RoboDK station: main for aircraft.rdk

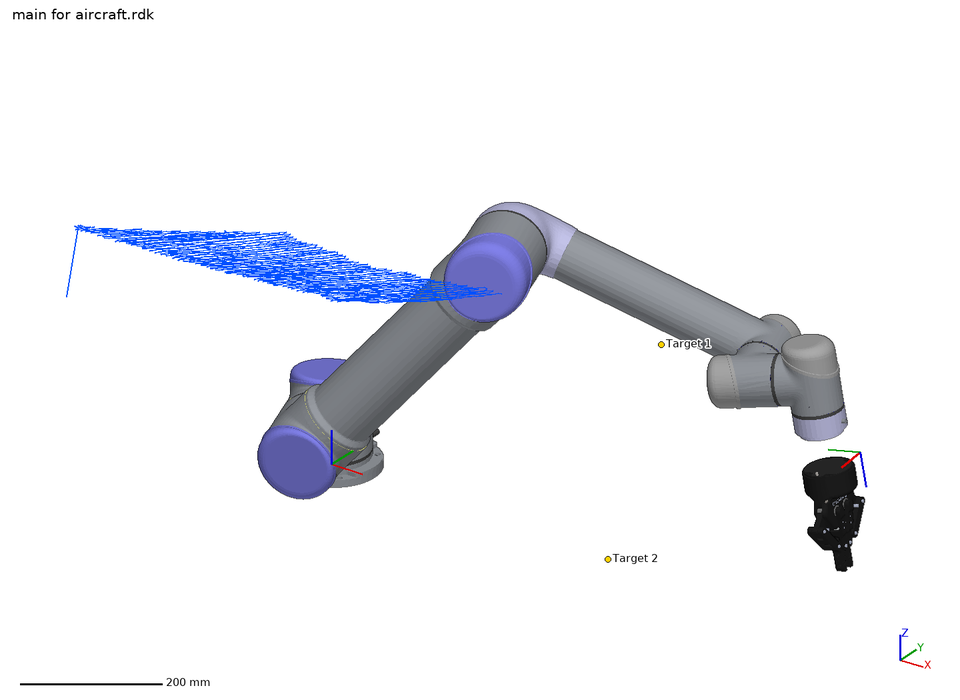
[picture v0: the station drawn from its stored meshes, robots at their saved joint values, targets as dots, program paths as lines]
Station main. Poses are relative to the parent item; angles as X-Y-Z fixed-axis rotations.
  - frame UR5 Base at (0, 0, 0) mm
    - robot UR5: 6 axes, payload 5 kg, reach 850 mm, repeatability 0.1 mm, weight 18.4 kg
        modified DH rows (alpha deg, a mm, theta deg, d mm): 0, 0, 0, 89.2; 90, 0, 180, 0; 0, 425, 0, 0; 0, 392.43, 0, 109; -90, 0, 0, 93.65; 90, 0, 180, 82
        joint limits [-360, -360, -360, -360, -360, -360] to [360, 360, 360, 360, 360, 360]; home [0, -90, -90, 0, 90, 0]; saved at [19.212, -130.821, -70.481, -59.3, 88.748, 13.688]
      - tool Gripper RobotiQ 85 Fully closed, TCP at (0, 0, 221.6) mm, size 121.5 x 75 x 160.2 mm
      - frame Object at (0, -58.4, 27.12) mm
        - object cloud_2 at (0, 0, 0) mm
    - target Target 1 (Cartesian target) at (643.45, -109, 411.64) mm, rotated rx -90 ry 0 rz -90 deg; joints [0, -90, -120, 30, 90, 0] of UR5
    - target Target 2 (Cartesian target) at (518.34, -61.08, 20.7) mm, rotated rx -149.99 ry -0.01 rz -84.67 deg; joints [5.34, -89.99, -135, -15, 89.99, 0] of UR5
  - machining project Path1 settings: rotZ(0) | rotX(0)*rotY(0) | rotZ(0)
  - program Path1 (2180 instructions, listed below)
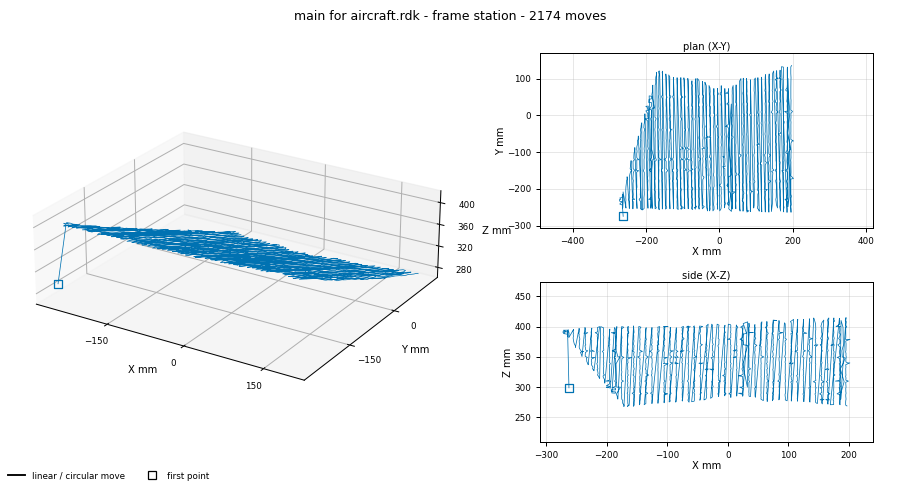
[picture p0: tool path of main for aircraft.rdk in frame station, 2174 of 2174 moves have a stored position in this frame; points joined in program order, loops and branches not executed]

--- program Path1 (robot UR5) ---
  Smooth(10)
  Set Ref.: UR5 Base
  Set Tool: Gripper RobotiQ 85 Fully closed
  Show Gripper RobotiQ 85 Fully closed
  Set speed (1000.0 mm/s)
  MoveJ 1 to (-262.02, -274.89, 298.94) mm, rotated rx -17.88 ry -1.25 rz 0.4 deg; joints [23.669, -136.733, -44.176, -77.159, 87.449, 17.927]
  MoveL 2 to (-262.02, -274.89, 298.94) mm, rotated rx -17.88 ry -1.25 rz 0.4 deg; joints [23.669, -136.733, -44.176, -77.159, 87.449, 17.927]
  MoveL 3 to (-264.31, -244.19, 394.09) mm, rotated rx -17.88 ry -1.25 rz 0.4 deg; joints [23.356, -142.512, -47.963, -67.579, 87.514, 17.62]
  MoveL 4 to (-264.31, -244.19, 394.09) mm, rotated rx -17.88 ry -1.25 rz 0.4 deg; joints [23.356, -142.512, -47.963, -67.579, 87.514, 17.62]
  Set speed (15.0 mm/s)
  MoveL 5 to (-271.37, -241.29, 394) mm, rotated rx -17.59 ry -0.18 rz 0.06 deg; joints [24.315, -142.277, -48.615, -67.291, 86.159, 18.561]
  MoveL 6 to (-265.21, -234.85, 391.18) mm, rotated rx -18.34 ry -0.72 rz 0.24 deg; joints [23.771, -141.372, -50.184, -67.121, 87.044, 18.065]
  MoveL 7 to (-271.75, -233.48, 391.83) mm, rotated rx -17.96 ry 0.25 rz -0.08 deg; joints [24.636, -141.351, -50.461, -66.885, 85.792, 18.911]
  MoveL 8 to (-271.9, -228.84, 390.33) mm, rotated rx -18.1 ry 0.31 rz -0.1 deg; joints [24.767, -140.701, -51.764, -66.391, 85.742, 19.05]
  MoveL 9 to (-268.61, -228.64, 390) mm, rotated rx -18.14 ry -0.12 rz 0.04 deg; joints [24.384, -140.498, -52.137, -66.09, 86.266, 18.666]
  MoveL 10 to (-271.13, -224.72, 388.5) mm, rotated rx -18.41 ry 0.27 rz -0.09 deg; joints [24.766, -140.169, -52.704, -66.263, 85.891, 19.068]
  MoveL 11 to (-264.69, -223.8, 387.46) mm, rotated rx -18.7 ry -0.08 rz 0.03 deg; joints [24.193, -139.886, -53.085, -66.288, 86.443, 18.513]
  MoveL 12 to (-264.01, -214.35, 383.52) mm, rotated rx -19.57 ry 0.41 rz -0.15 deg; joints [24.468, -138.955, -54.628, -66.688, 86.173, 18.846]
  MoveL 13 to (-263.28, -252.22, 395) mm, rotated rx -17 ry -2.06 rz 0.63 deg; joints [22.928, -142.903, -47.188, -66.845, 88.145, 17.134]
  MoveL 14 to (-261.82, -230.09, 389) mm, rotated rx -18.55 ry -0.65 rz 0.22 deg; joints [23.659, -140.571, -51.658, -66.67, 87.067, 17.969]
  MoveL 15 to (-262.24, -208.29, 381.79) mm, rotated rx -20.3 ry 0.18 rz -0.07 deg; joints [24.312, -138.465, -55.509, -66.903, 86.669, 18.726]
  MoveL 16 to (-254.38, -252.26, 395.31) mm, rotated rx -17.81 ry -2 rz 0.64 deg; joints [22.259, -143.318, -46.122, -68.265, 88.48, 16.534]
  MoveL 17 to (-254.85, -244.55, 394.03) mm, rotated rx -18.36 ry -1.42 rz 0.47 deg; joints [22.6, -142.604, -47.596, -68.221, 87.982, 16.907]
  MoveL 18 to (-255.09, -235.43, 390.85) mm, rotated rx -18.98 ry -1.16 rz 0.4 deg; joints [22.843, -141.518, -49.632, -67.954, 87.861, 17.185]
  MoveL 19 to (-254.54, -230.43, 389) mm, rotated rx -19.03 ry -1.01 rz 0.35 deg; joints [22.969, -140.693, -51.267, -67.243, 87.701, 17.314]
  MoveL 20 to (-255, -224.03, 387.47) mm, rotated rx -19.42 ry -0.43 rz 0.15 deg; joints [23.312, -140.084, -52.474, -67.22, 87.178, 17.681]
  MoveL 21 to (-254.65, -215.01, 384.18) mm, rotated rx -19.77 ry -0.12 rz 0.04 deg; joints [23.579, -138.889, -54.768, -66.567, 86.924, 17.968]
  MoveL 22 to (-255.09, -206.58, 381.26) mm, rotated rx -20.6 ry -0.07 rz 0.03 deg; joints [23.728, -138.168, -56.031, -66.846, 87.109, 18.159]
  MoveL 23 to (-254.81, -200.69, 379) mm, rotated rx -21.31 ry -0.04 rz 0.02 deg; joints [23.778, -137.716, -56.752, -67.264, 87.292, 18.244]
  MoveL 24 to (-254.51, -194.38, 376.76) mm, rotated rx -21.65 ry 0.05 rz -0.02 deg; joints [23.904, -136.986, -58.14, -66.963, 87.29, 18.385]
  MoveL 25 to (-253.55, -184.56, 372.52) mm, rotated rx -21.47 ry 0.4 rz -0.16 deg; joints [24.253, -135.357, -61.31, -65.393, 86.821, 18.729]
  MoveL 26 to (-252.52, -177.08, 370) mm, rotated rx -21.21 ry -0.12 rz 0.05 deg; joints [24.19, -134.062, -64.017, -63.546, 87.278, 18.645]
  MoveL 27 to (-251.17, -173.83, 368.17) mm, rotated rx -21.13 ry -0.62 rz 0.24 deg; joints [23.992, -133.403, -65.278, -62.689, 87.788, 18.438]
  MoveL 28 to (-251.35, -167.05, 365.62) mm, rotated rx -20.8 ry -1.05 rz 0.4 deg; joints [24.046, -132.249, -67.676, -60.989, 88.11, 18.47]
  MoveL 29 to (-245.27, -253.36, 397.1) mm, rotated rx -18.06 ry -1.59 rz 0.52 deg; joints [21.74, -143.678, -45.456, -68.922, 88.244, 16.045]
  MoveL 30 to (-244.89, -245.2, 395.32) mm, rotated rx -18.29 ry -1.31 rz 0.43 deg; joints [21.952, -142.513, -47.907, -67.941, 87.987, 16.269]
  MoveL 31 to (-244.93, -234.87, 391.11) mm, rotated rx -19.15 ry -0.83 rz 0.29 deg; joints [22.268, -141.35, -49.93, -68.065, 87.689, 16.633]
  MoveL 32 to (-245.96, -230.09, 389) mm, rotated rx -19.24 ry -1.01 rz 0.35 deg; joints [22.369, -140.564, -51.456, -67.362, 87.875, 16.735]
  MoveL 33 to (-245.08, -224.32, 387.67) mm, rotated rx -19.76 ry -0.9 rz 0.32 deg; joints [22.412, -140.052, -52.456, -67.409, 87.909, 16.806]
  MoveL 34 to (-245.41, -214.6, 384.46) mm, rotated rx -20.27 ry -0.68 rz 0.25 deg; joints [22.674, -138.901, -54.682, -66.904, 87.795, 17.093]
  MoveL 35 to (-244.36, -207.09, 381.36) mm, rotated rx -20.94 ry -0.36 rz 0.14 deg; joints [22.823, -138.135, -55.981, -67.109, 87.647, 17.276]
  MoveL 36 to (-244.03, -202.05, 379) mm, rotated rx -21.44 ry 0.03 rz -0.01 deg; joints [23.019, -137.675, -56.679, -67.493, 87.365, 17.499]
  MoveL 37 to (-245.13, -196.13, 376.68) mm, rotated rx -21.41 ry 0.07 rz -0.03 deg; joints [23.257, -136.756, -58.505, -66.575, 87.28, 17.733]
  MoveL 38 to (-244.73, -184.95, 372.15) mm, rotated rx -21.47 ry -0.36 rz 0.14 deg; joints [23.319, -135.037, -61.881, -64.841, 87.732, 17.792]
  MoveL 39 to (-244.68, -178.24, 370) mm, rotated rx -21.08 ry -0.66 rz 0.25 deg; joints [23.403, -133.845, -64.418, -63.026, 87.903, 17.853]
  MoveL 40 to (-245.12, -173.35, 367.97) mm, rotated rx -20.89 ry -0.84 rz 0.32 deg; joints [23.509, -133.026, -66.07, -61.958, 88.011, 17.946]
  MoveL 41 to (-244.93, -165.35, 364.68) mm, rotated rx -20.48 ry -1.14 rz 0.42 deg; joints [23.631, -131.646, -68.884, -60.034, 88.163, 18.042]
  MoveL 42 to (-243.12, -157.49, 361.29) mm, rotated rx -20.59 ry -1.28 rz 0.48 deg; joints [23.629, -130.568, -70.913, -59.139, 88.346, 18.045]
  MoveL 43 to (-240.83, -151.15, 358.5) mm, rotated rx -20.52 ry -0.67 rz 0.25 deg; joints [23.895, -129.668, -72.568, -58.54, 87.664, 18.312]
  MoveL 44 to (-238.06, -151.02, 358.75) mm, rotated rx -20.52 ry -0.37 rz 0.14 deg; joints [23.817, -129.648, -72.618, -58.609, 87.368, 18.239]
  MoveL 45 to (-243.08, -145.19, 357.68) mm, rotated rx -19.97 ry -0.57 rz 0.21 deg; joints [24.322, -128.85, -74.551, -56.9, 87.317, 18.705]
  MoveL 46 to (-241.78, -136.21, 354.56) mm, rotated rx -19.44 ry -0.13 rz 0.04 deg; joints [24.735, -127.521, -77.303, -55.15, 86.624, 19.09]
  MoveL 47 to (-240.49, -123.04, 350.5) mm, rotated rx -20.48 ry 0.16 rz -0.06 deg; joints [24.976, -126.522, -79.078, -55.474, 86.644, 19.392]
  MoveL 48 to (-235.56, -254.48, 398.54) mm, rotated rx -18.32 ry -2.03 rz 0.67 deg; joints [20.867, -143.917, -45.052, -69.191, 88.938, 15.202]
  MoveL 49 to (-234.99, -245.99, 396.5) mm, rotated rx -18.88 ry -1.71 rz 0.58 deg; joints [21.049, -142.919, -47.055, -68.812, 88.732, 15.413]
  MoveL 50 to (-234.59, -235.11, 391.54) mm, rotated rx -19.24 ry -1.1 rz 0.39 deg; joints [21.443, -141.197, -50.25, -67.874, 88.144, 15.824]
  MoveL 51 to (-237.42, -230.09, 389) mm, rotated rx -19.21 ry -0.91 rz 0.32 deg; joints [21.828, -140.327, -51.903, -67.134, 87.863, 16.203]
  MoveL 52 to (-230.9, -228.64, 390) mm, rotated rx -19.78 ry -0.55 rz 0.2 deg; joints [21.474, -140.556, -51.474, -67.979, 87.721, 15.887]
  MoveL 53 to (-235.09, -224.52, 387.67) mm, rotated rx -20 ry -0.49 rz 0.18 deg; joints [21.854, -140.039, -52.346, -67.868, 87.662, 16.273]
  MoveL 54 to (-234.47, -214.82, 383.61) mm, rotated rx -20.59 ry -0.14 rz 0.05 deg; joints [22.097, -138.831, -54.532, -67.568, 87.433, 16.545]
  MoveL 55 to (-235.27, -206.19, 381.33) mm, rotated rx -21.35 ry 0.02 rz -0.01 deg; joints [22.314, -138.126, -55.889, -67.709, 87.452, 16.796]
  MoveL 56 to (-234.79, -200.4, 379) mm, rotated rx -21.38 ry 0.17 rz -0.07 deg; joints [22.469, -137.224, -57.644, -66.937, 87.283, 16.952]
  MoveL 57 to (-234.99, -195.17, 376.66) mm, rotated rx -21.14 ry 0.11 rz -0.04 deg; joints [22.612, -136.221, -59.647, -65.694, 87.252, 17.082]
  MoveL 58 to (-235.1, -184.94, 371.79) mm, rotated rx -21.07 ry -0.25 rz 0.1 deg; joints [22.73, -134.526, -62.894, -63.969, 87.588, 17.192]
  MoveL 59 to (-234.21, -177.27, 370) mm, rotated rx -20.81 ry -0.51 rz 0.2 deg; joints [22.76, -133.36, -65.452, -62.243, 87.773, 17.206]
  MoveL 60 to (-235.54, -173.01, 368.33) mm, rotated rx -20.82 ry -0.65 rz 0.25 deg; joints [22.902, -132.788, -66.583, -61.655, 87.896, 17.345]
  MoveL 61 to (-234.9, -165.28, 365.2) mm, rotated rx -20.51 ry -0.38 rz 0.14 deg; joints [23.198, -131.55, -69.048, -60.228, 87.478, 17.626]
  MoveL 62 to (-234.35, -155.67, 361.24) mm, rotated rx -20.6 ry -0.05 rz 0.02 deg; joints [23.535, -130.314, -71.373, -59.352, 87.113, 17.968]
  MoveL 63 to (-231.01, -148.96, 360) mm, rotated rx -20.45 ry 0.48 rz -0.18 deg; joints [23.687, -129.488, -73.192, -58.398, 86.505, 18.121]
  MoveL 64 to (-234.82, -144.91, 357.2) mm, rotated rx -19.92 ry 0.4 rz -0.15 deg; joints [24.132, -128.646, -74.798, -57.136, 86.35, 18.534]
  MoveL 65 to (-235.11, -135.63, 354.57) mm, rotated rx -19.54 ry 0.45 rz -0.16 deg; joints [24.472, -127.421, -77.439, -55.389, 86.123, 18.849]
  MoveL 66 to (-235.19, -125.18, 350.94) mm, rotated rx -20.54 ry 0.28 rz -0.11 deg; joints [24.556, -126.657, -78.705, -55.788, 86.604, 18.982]
  MoveL 67 to (-231.56, -120.69, 349) mm, rotated rx -20.69 ry 0.55 rz -0.21 deg; joints [24.505, -126.104, -79.666, -55.613, 86.382, 18.945]
  MoveL 68 to (-233.13, -116.64, 348.05) mm, rotated rx -20.45 ry 0.78 rz -0.29 deg; joints [24.871, -125.628, -80.743, -54.885, 86.02, 19.3]
  MoveL 69 to (-232.48, -103.36, 342.04) mm, rotated rx -19.32 ry 1.44 rz -0.51 deg; joints [25.695, -123.513, -84.948, -52.026, 84.852, 20.074]
  MoveL 70 to (-230.44, -93.33, 338) mm, rotated rx -18.72 ry 1.77 rz -0.6 deg; joints [26.094, -122.086, -87.812, -50.172, 84.258, 20.443]
  MoveL 71 to (-230.35, -87.47, 337) mm, rotated rx -18.21 ry 1.44 rz -0.47 deg; joints [26.189, -121.353, -89.619, -48.515, 84.393, 20.494]
  MoveL 72 to (-224.26, -253.51, 397.45) mm, rotated rx -17.86 ry -0.84 rz 0.27 deg; joints [20.624, -143.106, -46.589, -68.346, 87.657, 14.95]
  MoveL 73 to (-224.65, -244.82, 394.97) mm, rotated rx -19.31 ry -0.98 rz 0.34 deg; joints [20.617, -142.743, -47.048, -69.609, 88.186, 15.016]
  MoveL 74 to (-225.29, -234.71, 391.92) mm, rotated rx -20.17 ry -0.81 rz 0.3 deg; joints [20.831, -141.712, -49, -69.577, 88.204, 15.269]
  MoveL 75 to (-225.48, -228.49, 390.54) mm, rotated rx -20.35 ry -0.34 rz 0.13 deg; joints [21.123, -140.916, -50.662, -69.025, 87.722, 15.57]
  MoveL 76 to (-224.94, -222.92, 387.64) mm, rotated rx -20.71 ry 0.23 rz -0.09 deg; joints [21.393, -140.188, -51.88, -69.062, 87.189, 15.86]
  MoveL 77 to (-225.17, -214.13, 383.95) mm, rotated rx -20.79 ry 0.57 rz -0.22 deg; joints [21.72, -138.779, -54.606, -67.933, 86.818, 16.192]
  MoveL 78 to (-225.18, -205.91, 381.59) mm, rotated rx -21.52 ry 0.54 rz -0.21 deg; joints [21.803, -138.055, -55.982, -67.985, 87.037, 16.303]
  MoveL 79 to (-225.62, -200.65, 379) mm, rotated rx -21.32 ry 0.54 rz -0.21 deg; joints [21.976, -137.033, -57.975, -66.831, 86.957, 16.468]
  MoveL 80 to (-224.43, -195.01, 376.66) mm, rotated rx -20.83 ry 0.36 rz -0.14 deg; joints [22.001, -135.783, -60.553, -64.972, 87.004, 16.468]
  MoveL 81 to (-225.11, -184.75, 371.86) mm, rotated rx -20.72 ry 0 rz 0 deg; joints [22.159, -134.102, -63.794, -63.21, 87.314, 16.615]
  MoveL 82 to (-225.01, -176.36, 370) mm, rotated rx -20.72 ry -0.1 rz 0.04 deg; joints [22.292, -133.055, -66.07, -61.953, 87.394, 16.744]
  MoveL 83 to (-224.73, -171.97, 369) mm, rotated rx -20.69 ry -0.13 rz 0.05 deg; joints [22.359, -132.502, -67.271, -61.275, 87.406, 16.809]
  MoveL 84 to (-225.03, -164.63, 365.7) mm, rotated rx -20.72 ry -0.05 rz 0.02 deg; joints [22.594, -131.478, -69.194, -60.433, 87.292, 17.044]
  MoveL 85 to (-225.2, -154.48, 361.68) mm, rotated rx -20.84 ry 0.43 rz -0.16 deg; joints [23.042, -130.232, -71.548, -59.619, 86.778, 17.501]
  MoveL 86 to (-220.05, -150.42, 359) mm, rotated rx -20.71 ry 0.42 rz -0.16 deg; joints [22.786, -129.405, -73, -58.855, 86.781, 17.241]
  MoveL 87 to (-226.78, -148.96, 360) mm, rotated rx -20.5 ry 0.65 rz -0.24 deg; joints [23.434, -129.436, -73.256, -58.471, 86.387, 17.877]
  MoveL 88 to (-224.77, -144.73, 357.84) mm, rotated rx -19.94 ry 0.76 rz -0.28 deg; joints [23.52, -128.522, -75.092, -57.056, 86.088, 17.936]
  MoveL 89 to (-224.77, -135.41, 353.91) mm, rotated rx -19.75 ry 0.67 rz -0.24 deg; joints [23.757, -127.226, -77.611, -55.638, 86.088, 18.159]
  MoveL 90 to (-224.84, -125.83, 350.62) mm, rotated rx -20.41 ry 0.59 rz -0.22 deg; joints [23.895, -126.414, -79.062, -55.616, 86.355, 18.328]
  MoveL 91 to (-224.94, -120.84, 349) mm, rotated rx -20.56 ry 0.48 rz -0.18 deg; joints [23.972, -125.908, -80.054, -55.237, 86.496, 18.409]
  MoveL 92 to (-219.39, -120.69, 349) mm, rotated rx -20.26 ry 0.42 rz -0.15 deg; joints [23.551, -125.645, -80.641, -54.588, 86.535, 17.977]
  MoveL 93 to (-224.89, -115.22, 346.52) mm, rotated rx -20.17 ry 0.44 rz -0.16 deg; joints [24.165, -125.019, -81.828, -53.98, 86.386, 18.579]
  MoveL 94 to (-225.08, -104.78, 342.27) mm, rotated rx -19.57 ry 0.5 rz -0.18 deg; joints [24.6, -123.516, -84.849, -51.942, 86.062, 18.979]
  MoveL 95 to (-224.21, -97.29, 340.35) mm, rotated rx -19.46 ry 0.37 rz -0.13 deg; joints [24.7, -122.698, -86.622, -50.846, 86.135, 19.068]
  MoveL 96 to (-224.95, -92.6, 338.54) mm, rotated rx -18.94 ry 0.42 rz -0.14 deg; joints [25.004, -121.973, -88.173, -49.565, 85.866, 19.339]
  MoveL 97 to (-224.77, -85.07, 336.69) mm, rotated rx -18.19 ry 0.24 rz -0.08 deg; joints [25.243, -120.953, -90.57, -47.436, 85.753, 19.523]
  MoveL 98 to (-222.4, -76.14, 333.17) mm, rotated rx -18.45 ry 0.43 rz -0.14 deg; joints [25.382, -120.026, -92.205, -47.047, 85.625, 19.681]
  MoveL 99 to (-223.06, -68.06, 330) mm, rotated rx -18.49 ry 1.06 rz -0.36 deg; joints [26, -119.213, -93.672, -46.709, 84.9, 20.313]
  MoveL 100 to (-221.63, -65.81, 329) mm, rotated rx -18.73 ry 1.11 rz -0.38 deg; joints [25.943, -119.016, -93.931, -46.884, 84.938, 20.273]
  MoveL 101 to (-220.78, -56, 327) mm, rotated rx -18.67 ry 1.16 rz -0.39 deg; joints [26.21, -118.144, -95.917, -45.753, 84.829, 20.534]
  MoveL 102 to (-211.47, -256.98, 400) mm, rotated rx -17.76 ry -0.5 rz 0.16 deg; joints [19.817, -143.56, -45.828, -68.607, 87.461, 14.158]
  MoveL 103 to (-215.08, -253.73, 398.33) mm, rotated rx -17.78 ry -0.23 rz 0.07 deg; joints [20.226, -143.02, -46.84, -68.247, 87.108, 14.562]
  MoveL 104 to (-215.14, -245.39, 395.51) mm, rotated rx -19.28 ry -0.34 rz 0.12 deg; joints [20.202, -142.704, -47.117, -69.707, 87.607, 14.612]
  MoveL 105 to (-214.75, -234.66, 391.28) mm, rotated rx -20.45 ry -0.22 rz 0.08 deg; joints [20.317, -141.664, -48.87, -70.166, 87.762, 14.779]
  MoveL 106 to (-218.67, -228.64, 390) mm, rotated rx -20.94 ry -0.18 rz 0.07 deg; joints [20.661, -141.183, -49.867, -70.146, 87.791, 15.14]
  MoveL 107 to (-214.54, -223.91, 387.58) mm, rotated rx -21.55 ry -0.05 rz 0.02 deg; joints [20.471, -140.68, -50.618, -70.524, 87.839, 14.977]
  MoveL 108 to (-215.61, -214.66, 384.5) mm, rotated rx -21.1 ry 0.71 rz -0.28 deg; joints [21.068, -138.926, -54.253, -68.45, 86.849, 15.562]
  MoveL 109 to (-214.44, -207.03, 381.09) mm, rotated rx -21.27 ry 0.96 rz -0.37 deg; joints [21.23, -137.749, -56.466, -67.65, 86.618, 15.733]
  MoveL 110 to (-214.86, -202.28, 378.8) mm, rotated rx -21.02 ry 0.81 rz -0.31 deg; joints [21.332, -136.774, -58.4, -66.412, 86.691, 15.821]
  MoveL 111 to (-215.13, -195.25, 376.54) mm, rotated rx -20.48 ry 0.52 rz -0.2 deg; joints [21.441, -135.394, -61.348, -64.252, 86.821, 15.901]
  MoveL 112 to (-215.18, -184.32, 372.5) mm, rotated rx -20.33 ry 0 rz 0 deg; joints [21.486, -133.693, -64.797, -62.208, 87.312, 15.932]
  MoveL 113 to (-214.76, -177.32, 370.1) mm, rotated rx -20.58 ry -0.24 rz 0.09 deg; joints [21.482, -132.86, -66.429, -61.573, 87.629, 15.935]
  MoveL 114 to (-214.8, -172.7, 368.5) mm, rotated rx -20.62 ry -0.28 rz 0.11 deg; joints [21.566, -132.265, -67.615, -61.017, 87.666, 16.02]
  MoveL 115 to (-215.35, -164.89, 365.18) mm, rotated rx -20.82 ry -0.22 rz 0.08 deg; joints [21.793, -131.294, -69.413, -60.406, 87.624, 16.253]
  MoveL 116 to (-215.08, -155.84, 361.5) mm, rotated rx -21.27 ry 0.01 rz 0 deg; joints [22.033, -130.327, -71.135, -60.165, 87.476, 16.514]
  MoveL 117 to (-214.17, -150.56, 358.58) mm, rotated rx -20.81 ry -0.02 rz 0.01 deg; joints [22.144, -129.276, -73.162, -58.746, 87.359, 16.603]
  MoveL 118 to (-214.93, -145.12, 357.5) mm, rotated rx -20.02 ry 0.14 rz -0.05 deg; joints [22.486, -128.318, -75.399, -56.772, 86.918, 16.906]
  MoveL 119 to (-215.06, -135.25, 353.84) mm, rotated rx -19.81 ry 0.4 rz -0.14 deg; joints [22.884, -127.028, -77.963, -55.407, 86.526, 17.295]
  MoveL 120 to (-215.16, -125.02, 350.6) mm, rotated rx -20.24 ry 0.34 rz -0.12 deg; joints [23.071, -126.058, -79.834, -54.9, 86.685, 17.499]
  MoveL 121 to (-215.14, -115.54, 346.98) mm, rotated rx -19.7 ry -0.22 rz 0.08 deg; joints [23.146, -124.657, -82.738, -52.716, 87.077, 17.536]
  MoveL 122 to (-215.06, -104.83, 341.87) mm, rotated rx -19.58 ry -0.68 rz 0.24 deg; joints [23.253, -123.215, -85.418, -51.211, 87.489, 17.628]
  MoveL 123 to (-215.04, -95.66, 340.39) mm, rotated rx -19.52 ry -0.81 rz 0.29 deg; joints [23.435, -122.375, -87.412, -49.966, 87.561, 17.802]
  MoveL 124 to (-216.04, -91.06, 339) mm, rotated rx -19.13 ry -0.74 rz 0.26 deg; joints [23.732, -121.767, -88.759, -48.9, 87.32, 18.074]
  MoveL 125 to (-215.04, -84.65, 335.85) mm, rotated rx -18.47 ry -0.55 rz 0.18 deg; joints [24.037, -120.705, -90.866, -47.3, 86.86, 18.337]
  MoveL 126 to (-215.15, -74.93, 332.53) mm, rotated rx -18.88 ry 0.01 rz -0.01 deg; joints [24.543, -119.876, -92.321, -47.29, 86.337, 18.871]
  MoveL 127 to (-214.17, -67.84, 330.28) mm, rotated rx -19.3 ry 0.73 rz -0.25 deg; joints [24.954, -119.34, -93.221, -47.592, 85.686, 19.319]
  MoveL 128 to (-215.65, -63.24, 328.81) mm, rotated rx -19.02 ry 1.07 rz -0.37 deg; joints [25.433, -118.823, -94.323, -46.905, 85.176, 19.785]
  MoveL 129 to (-214.55, -54.89, 326.32) mm, rotated rx -18.36 ry 1.15 rz -0.38 deg; joints [25.761, -117.761, -96.683, -45.034, 84.807, 20.07]
  MoveL 130 to (-213.92, -45.69, 322.33) mm, rotated rx -18.33 ry 0.81 rz -0.27 deg; joints [25.871, -116.693, -98.64, -44.003, 85.113, 20.166]
  MoveL 131 to (-214.96, -38.18, 320) mm, rotated rx -18.64 ry 1.1 rz -0.37 deg; joints [26.313, -116.121, -99.68, -43.979, 84.855, 20.633]
  MoveL 132 to (-213.6, -33.58, 318.68) mm, rotated rx -18.78 ry 0.99 rz -0.34 deg; joints [26.269, -115.713, -100.481, -43.671, 85.023, 20.594]
  MoveL 133 to (-212.85, -26.02, 317.07) mm, rotated rx -19.11 ry 0.76 rz -0.26 deg; joints [26.28, -115.177, -101.632, -43.28, 85.364, 20.619]
  MoveL 134 to (-211.34, -19.96, 314) mm, rotated rx -18.89 ry 0.62 rz -0.21 deg; joints [26.35, -114.349, -103.112, -42.378, 85.411, 20.67]
  MoveL 135 to (-209.64, -257.5, 400) mm, rotated rx -17.8 ry -0.77 rz 0.25 deg; joints [19.583, -143.605, -45.709, -68.642, 87.787, 13.928]
  MoveL 136 to (-204.95, -253.35, 398) mm, rotated rx -18.23 ry -1.18 rz 0.39 deg; joints [19.149, -142.99, -46.782, -68.488, 88.401, 13.521]
  MoveL 137 to (-204.97, -245.48, 396.69) mm, rotated rx -19.72 ry -0.8 rz 0.29 deg; joints [19.286, -142.956, -46.663, -70.186, 88.347, 13.726]
  MoveL 138 to (-205.03, -235.25, 392.46) mm, rotated rx -20.38 ry -0.68 rz 0.25 deg; joints [19.462, -141.576, -49.209, -69.692, 88.359, 13.928]
  MoveL 139 to (-205.43, -224.42, 387.26) mm, rotated rx -21.93 ry -0.36 rz 0.15 deg; joints [19.681, -140.783, -50.245, -71.043, 88.373, 14.205]
  MoveL 140 to (-204.52, -215.24, 383.39) mm, rotated rx -21.97 ry 0.17 rz -0.07 deg; joints [19.999, -139.225, -53.255, -69.79, 87.787, 14.527]
  MoveL 141 to (-204.64, -208.09, 380.47) mm, rotated rx -21.43 ry 0.52 rz -0.21 deg; joints [20.343, -137.675, -56.419, -67.76, 87.232, 14.853]
  MoveL 142 to (-205.04, -203.35, 378.95) mm, rotated rx -20.84 ry 0.64 rz -0.24 deg; joints [20.57, -136.581, -58.772, -65.973, 86.928, 15.056]
  MoveL 143 to (-204.88, -196.28, 376.63) mm, rotated rx -20.12 ry 0.53 rz -0.2 deg; joints [20.729, -135.088, -61.977, -63.541, 86.83, 15.182]
  MoveL 144 to (-205, -185.03, 371.9) mm, rotated rx -19.72 ry -0.15 rz 0.05 deg; joints [20.744, -133.143, -65.896, -60.99, 87.419, 15.169]
  MoveL 145 to (-205.03, -177.27, 370) mm, rotated rx -20.21 ry -0.51 rz 0.19 deg; joints [20.697, -132.444, -67.326, -60.631, 87.934, 15.141]
  MoveL 146 to (-204.93, -172.76, 368.52) mm, rotated rx -20.68 ry -0.65 rz 0.24 deg; joints [20.678, -132.107, -67.911, -60.798, 88.198, 15.141]
  MoveL 147 to (-204.82, -165.16, 364.5) mm, rotated rx -21.02 ry -0.39 rz 0.15 deg; joints [20.916, -131.16, -69.481, -60.589, 87.99, 15.393]
  MoveL 148 to (-204.5, -155.71, 360.94) mm, rotated rx -21.24 ry -0.51 rz 0.2 deg; joints [21.028, -130.018, -71.669, -59.724, 88.152, 15.512]
  MoveL 149 to (-206.82, -150.79, 359) mm, rotated rx -20.95 ry -0.5 rz 0.19 deg; joints [21.351, -129.256, -73.23, -58.653, 88.019, 15.819]
  MoveL 150 to (-204.93, -144.78, 356.58) mm, rotated rx -20.14 ry -0.63 rz 0.23 deg; joints [21.386, -128.028, -75.828, -56.468, 87.923, 15.816]
  MoveL 151 to (-205.04, -134.95, 353.15) mm, rotated rx -19.96 ry -0.77 rz 0.28 deg; joints [21.584, -126.753, -78.422, -54.938, 87.983, 16.001]
  MoveL 152 to (-204.99, -125.88, 350.85) mm, rotated rx -20.02 ry -1.07 rz 0.39 deg; joints [21.65, -125.802, -80.464, -53.82, 88.287, 16.067]
  MoveL 153 to (-205.26, -120.69, 349) mm, rotated rx -19.54 ry -1.15 rz 0.41 deg; joints [21.822, -124.984, -82.218, -52.407, 88.205, 16.211]
  MoveL 154 to (-204.58, -114.95, 346.71) mm, rotated rx -19.32 ry -1.28 rz 0.45 deg; joints [21.881, -124.188, -83.82, -51.347, 88.268, 16.256]
  MoveL 155 to (-205.2, -105.09, 342.08) mm, rotated rx -19.68 ry -1.24 rz 0.44 deg; joints [22.168, -123.113, -85.622, -50.99, 88.279, 16.558]
  MoveL 156 to (-204.45, -96.61, 340.14) mm, rotated rx -19.5 ry -0.88 rz 0.31 deg; joints [22.509, -122.224, -87.57, -49.883, 87.796, 16.888]
  MoveL 157 to (-205.05, -91.23, 338.14) mm, rotated rx -19.32 ry -0.8 rz 0.28 deg; joints [22.769, -121.564, -88.894, -49.084, 87.614, 17.135]
  MoveL 158 to (-204.47, -84.21, 334.84) mm, rotated rx -18.96 ry -0.4 rz 0.14 deg; joints [23.167, -120.575, -90.748, -48.022, 87.027, 17.513]
  MoveL 159 to (-204.89, -74.93, 332.14) mm, rotated rx -19.34 ry 0.34 rz -0.12 deg; joints [23.762, -119.84, -92.11, -48.027, 86.289, 18.135]
  MoveL 160 to (-204.93, -67.67, 330.35) mm, rotated rx -19.58 ry 0.35 rz -0.13 deg; joints [23.941, -119.264, -93.299, -47.666, 86.324, 18.325]
  MoveL 161 to (-205.03, -62.07, 328.65) mm, rotated rx -18.82 ry 0.08 rz -0.03 deg; joints [24.097, -118.414, -95.267, -45.737, 86.338, 18.43]
  MoveL 162 to (-205.07, -54.88, 326.09) mm, rotated rx -18.28 ry 0.06 rz -0.02 deg; joints [24.403, -117.481, -97.258, -44.182, 86.124, 18.698]
  MoveL 163 to (-205.04, -44.7, 321.78) mm, rotated rx -18.6 ry 0.26 rz -0.09 deg; joints [24.792, -116.476, -98.936, -43.908, 85.955, 19.105]
  MoveL 164 to (-203.28, -37.8, 320.14) mm, rotated rx -19 ry 0.05 rz -0.02 deg; joints [24.677, -115.979, -99.929, -43.712, 86.316, 19.011]
  MoveL 165 to (-205.78, -33.38, 318.45) mm, rotated rx -19.04 ry 0.16 rz -0.05 deg; joints [25.101, -115.578, -100.66, -43.485, 86.147, 19.435]
  MoveL 166 to (-205.25, -24.93, 316.02) mm, rotated rx -19.15 ry 0.07 rz -0.02 deg; joints [25.273, -114.829, -102.182, -42.795, 86.237, 19.609]
  MoveL 167 to (-203.31, -15.98, 312.57) mm, rotated rx -19.01 ry 0.66 rz -0.23 deg; joints [25.746, -113.849, -103.984, -42.084, 85.523, 20.082]
  MoveL 168 to (-203.18, -4.3, 308) mm, rotated rx -18.97 ry 1.38 rz -0.47 deg; joints [26.569, -112.659, -106.108, -41.442, 84.648, 20.916]
  MoveL 169 to (-202.82, 4.49, 306.61) mm, rotated rx -18.29 ry 0.81 rz -0.27 deg; joints [26.668, -111.789, -108.423, -39.155, 84.955, 20.95]
  MoveL 170 to (-194.49, -252.71, 395.77) mm, rotated rx -18.72 ry -1.54 rz 0.52 deg; joints [18.28, -142.815, -46.713, -69.104, 89.066, 12.691]
  MoveL 171 to (-194.73, -245.58, 395.76) mm, rotated rx -20.04 ry -1.53 rz 0.56 deg; joints [18.287, -142.877, -46.628, -70.41, 89.354, 12.752]
  MoveL 172 to (-194.89, -235.56, 393.15) mm, rotated rx -20.8 ry -1.3 rz 0.49 deg; joints [18.48, -141.803, -48.749, -70.162, 89.259, 12.972]
  MoveL 173 to (-194.93, -223.93, 387.29) mm, rotated rx -22.28 ry -0.81 rz 0.33 deg; joints [18.754, -140.769, -50.227, -71.281, 89.058, 13.295]
  MoveL 174 to (-195.26, -215.5, 383.83) mm, rotated rx -22.28 ry -0.6 rz 0.25 deg; joints [19.01, -139.305, -53.099, -69.929, 88.804, 13.551]
  MoveL 175 to (-195.8, -208.58, 380.5) mm, rotated rx -21.68 ry -0.52 rz 0.21 deg; joints [19.268, -137.67, -56.384, -67.722, 88.54, 13.786]
  MoveL 176 to (-194.51, -203.7, 378.38) mm, rotated rx -21.11 ry -0.59 rz 0.23 deg; joints [19.295, -136.464, -58.876, -65.87, 88.47, 13.793]
  MoveL 177 to (-194.92, -195.07, 376.58) mm, rotated rx -19.92 ry -0.18 rz 0.07 deg; joints [19.758, -134.623, -63.03, -62.527, 87.681, 14.205]
  MoveL 178 to (-195.2, -184.4, 372.39) mm, rotated rx -19.27 ry -0.36 rz 0.12 deg; joints [19.988, -132.713, -66.975, -59.818, 87.655, 14.401]
  MoveL 179 to (-194.53, -176.53, 370.07) mm, rotated rx -19.83 ry -0.63 rz 0.23 deg; joints [19.92, -131.997, -68.35, -59.625, 88.092, 14.357]
  MoveL 180 to (-195.99, -172.09, 368.31) mm, rotated rx -20.47 ry -0.86 rz 0.32 deg; joints [19.958, -131.752, -68.662, -60.119, 88.484, 14.42]
  MoveL 181 to (-194.94, -165.13, 365.13) mm, rotated rx -21.02 ry -1.17 rz 0.45 deg; joints [19.839, -131.03, -69.872, -60.077, 88.962, 14.323]
  MoveL 182 to (-195.09, -155.17, 361.78) mm, rotated rx -20.9 ry -1.41 rz 0.54 deg; joints [19.962, -129.694, -72.609, -58.493, 89.162, 14.438]
  MoveL 183 to (-195.21, -144.9, 357.09) mm, rotated rx -20.16 ry -1.61 rz 0.59 deg; joints [20.194, -127.916, -76.174, -55.939, 89.136, 14.635]
  MoveL 184 to (-195.12, -135.4, 353.81) mm, rotated rx -19.64 ry -1.39 rz 0.5 deg; joints [20.551, -126.542, -79.031, -54.025, 88.71, 14.963]
  MoveL 185 to (-195.08, -125.88, 351.05) mm, rotated rx -19.85 ry -1.39 rz 0.5 deg; joints [20.731, -125.593, -80.951, -53.266, 88.737, 15.151]
  MoveL 186 to (-194.49, -120.69, 349) mm, rotated rx -19.68 ry -1.32 rz 0.47 deg; joints [20.862, -124.885, -82.353, -52.432, 88.588, 15.273]
  MoveL 187 to (-194.92, -114.33, 346.48) mm, rotated rx -19.49 ry -1.14 rz 0.4 deg; joints [21.156, -124.055, -83.98, -51.509, 88.298, 15.554]
  MoveL 188 to (-194.89, -104.22, 343.1) mm, rotated rx -20 ry -0.98 rz 0.36 deg; joints [21.408, -123.162, -85.607, -51.315, 88.233, 15.828]
  MoveL 189 to (-195.3, -95.28, 340.8) mm, rotated rx -19.95 ry -0.73 rz 0.27 deg; joints [21.779, -122.265, -87.516, -50.342, 87.902, 16.193]
  MoveL 190 to (-193.62, -90.85, 339) mm, rotated rx -19.75 ry -0.49 rz 0.17 deg; joints [21.896, -121.656, -88.697, -49.662, 87.577, 16.302]
  MoveL 191 to (-195.07, -84.79, 336.78) mm, rotated rx -19.55 ry -0.21 rz 0.07 deg; joints [22.339, -120.938, -90.127, -48.861, 87.161, 16.732]
  MoveL 192 to (-194.89, -74.97, 332.28) mm, rotated rx -19.58 ry 0.28 rz -0.1 deg; joints [22.84, -119.794, -92.117, -48.227, 86.582, 17.237]
  MoveL 193 to (-195.34, -67.92, 330.04) mm, rotated rx -19.19 ry 0.27 rz -0.09 deg; joints [23.124, -118.932, -93.964, -46.873, 86.435, 17.496]
  MoveL 194 to (-194.8, -62.59, 328.36) mm, rotated rx -18.63 ry 0.19 rz -0.07 deg; joints [23.277, -118.187, -95.633, -45.409, 86.312, 17.614]
  MoveL 195 to (-195.02, -54.65, 325.09) mm, rotated rx -18.39 ry 0.42 rz -0.14 deg; joints [23.694, -117.236, -97.447, -44.416, 85.929, 18.015]
  MoveL 196 to (-194.94, -44.81, 321.8) mm, rotated rx -18.54 ry 0.61 rz -0.21 deg; joints [24.066, -116.314, -99.197, -43.82, 85.715, 18.395]
  MoveL 197 to (-195.07, -37.32, 320.37) mm, rotated rx -18.99 ry 0.35 rz -0.12 deg; joints [24.095, -115.856, -100.191, -43.626, 86.114, 18.443]
  MoveL 198 to (-194.89, -32.21, 318.3) mm, rotated rx -19.17 ry 0.23 rz -0.08 deg; joints [24.157, -115.361, -101.04, -43.401, 86.283, 18.512]
  MoveL 199 to (-194.91, -24.98, 315.17) mm, rotated rx -19.36 ry 0.28 rz -0.1 deg; joints [24.4, -114.63, -102.257, -43.127, 86.253, 18.764]
  MoveL 200 to (-195.11, -15.18, 311.61) mm, rotated rx -19.14 ry 0.67 rz -0.23 deg; joints [24.998, -113.586, -104.268, -42.129, 85.688, 19.351]
  MoveL 201 to (-201.2, -9.33, 310) mm, rotated rx -19.28 ry 1.02 rz -0.36 deg; joints [25.937, -113.23, -104.985, -42.098, 85.222, 20.298]
  MoveL 202 to (-193.53, -8.51, 310) mm, rotated rx -19.2 ry 0.65 rz -0.23 deg; joints [25.051, -113.021, -105.471, -41.553, 85.716, 19.407]
  MoveL 203 to (-195.01, -3.37, 307.67) mm, rotated rx -18.82 ry 0.44 rz -0.15 deg; joints [25.341, -112.342, -106.811, -40.476, 85.753, 19.665]
  MoveL 204 to (-194.99, 5.48, 305.33) mm, rotated rx -18.19 ry 0.23 rz -0.08 deg; joints [25.659, -111.387, -109.049, -38.547, 85.686, 19.932]
  MoveL 205 to (-200.33, 12.39, 302.33) mm, rotated rx -18.09 ry -0.06 rz 0.02 deg; joints [26.325, -110.699, -110.322, -37.813, 85.812, 20.573]
  MoveL 206 to (-194.51, 14, 301.44) mm, rotated rx -18.01 ry 0.15 rz -0.05 deg; joints [25.95, -110.383, -110.828, -37.594, 85.644, 20.204]
  MoveL 207 to (-196.3, 22.05, 300) mm, rotated rx -18 ry 0.12 rz -0.04 deg; joints [26.408, -109.832, -112.197, -36.785, 85.585, 20.653]
  MoveL 208 to (-200.35, 24.84, 300) mm, rotated rx -17.83 ry 0.13 rz -0.04 deg; joints [26.956, -109.728, -112.699, -36.28, 85.406, 21.18]
  MoveL 209 to (-193.61, 25.7, 298.55) mm, rotated rx -17.9 ry 0.59 rz -0.19 deg; joints [26.578, -109.403, -112.942, -36.57, 85.048, 20.827]
  MoveL 210 to (-186.95, -252.68, 398.44) mm, rotated rx -18.8 ry -1.22 rz 0.41 deg; joints [17.864, -143.084, -46.503, -69.184, 88.829, 12.286]
  MoveL 211 to (-185.88, -245.71, 397.19) mm, rotated rx -20.05 ry -1.18 rz 0.43 deg; joints [17.802, -142.946, -46.644, -70.404, 89.081, 12.276]
  MoveL 212 to (-184.86, -235.76, 393.22) mm, rotated rx -20.75 ry -1.32 rz 0.5 deg; joints [17.781, -141.64, -49.068, -69.945, 89.386, 12.28]
  MoveL 213 to (-185.08, -228.71, 390.11) mm, rotated rx -21.83 ry -1.49 rz 0.6 deg; joints [17.758, -141.172, -49.698, -70.789, 89.802, 12.293]
  MoveL 214 to (-192.16, -228.64, 390) mm, rotated rx -21.65 ry -1.19 rz 0.47 deg; joints [18.382, -141.139, -49.786, -70.64, 89.358, 12.905]
  MoveL 215 to (-184.84, -223.44, 388.16) mm, rotated rx -22.73 ry -1.37 rz 0.57 deg; joints [17.797, -140.965, -49.906, -71.697, 89.873, 12.359]
  MoveL 216 to (-184.78, -215.5, 384.84) mm, rotated rx -22.3 ry -1.15 rz 0.47 deg; joints [18.051, -139.236, -53.395, -69.57, 89.507, 12.598]
  MoveL 217 to (-185.13, -203.61, 377.72) mm, rotated rx -21.35 ry -1.07 rz 0.42 deg; joints [18.416, -136.371, -58.922, -66.005, 89.157, 12.929]
  MoveL 218 to (-184.93, -195.05, 376.32) mm, rotated rx -20.56 ry -0.72 rz 0.27 deg; joints [18.755, -134.807, -62.471, -63.353, 88.554, 13.238]
  MoveL 219 to (-184.93, -184.74, 373.35) mm, rotated rx -19.09 ry -0.39 rz 0.14 deg; joints [19.215, -132.607, -67.347, -59.339, 87.789, 13.633]
  MoveL 220 to (-185.37, -177.08, 370.39) mm, rotated rx -19.31 ry -0.62 rz 0.22 deg; joints [19.279, -131.679, -69.12, -58.656, 88.069, 13.703]
  MoveL 221 to (-184.65, -172.48, 368.65) mm, rotated rx -19.82 ry -0.78 rz 0.28 deg; joints [19.198, -131.322, -69.685, -58.902, 88.37, 13.644]
  MoveL 222 to (-185.19, -164.73, 365.76) mm, rotated rx -20.68 ry -0.99 rz 0.38 deg; joints [19.214, -130.759, -70.58, -59.35, 88.796, 13.693]
  MoveL 223 to (-185, -154.78, 362.5) mm, rotated rx -20.57 ry -1.29 rz 0.48 deg; joints [19.279, -129.442, -73.295, -57.763, 89.058, 13.752]
  MoveL 224 to (-190.55, -148.96, 360) mm, rotated rx -20.55 ry -1.74 rz 0.65 deg; joints [19.634, -128.712, -74.734, -56.922, 89.464, 14.099]
  MoveL 225 to (-185.08, -143.52, 357.79) mm, rotated rx -20.23 ry -1.73 rz 0.64 deg; joints [19.361, -127.787, -76.59, -55.682, 89.417, 13.817]
  MoveL 226 to (-185.16, -135.12, 354.37) mm, rotated rx -20.24 ry -1.32 rz 0.49 deg; joints [19.724, -126.743, -78.543, -54.898, 88.943, 14.177]
  MoveL 227 to (-184.67, -125.32, 351.06) mm, rotated rx -19.83 ry -0.81 rz 0.29 deg; joints [20.174, -125.423, -81.246, -53.267, 88.231, 14.605]
  MoveL 228 to (-187.47, -120.69, 349) mm, rotated rx -19.84 ry -0.84 rz 0.3 deg; joints [20.494, -124.878, -82.255, -52.815, 88.205, 14.921]
  MoveL 229 to (-184.94, -114.44, 347.18) mm, rotated rx -19.85 ry -0.46 rz 0.17 deg; joints [20.599, -124.192, -83.635, -52.24, 87.803, 15.029]
  MoveL 230 to (-185.16, -104.68, 344.2) mm, rotated rx -19.8 ry -0.32 rz 0.11 deg; joints [20.915, -123.129, -85.813, -51.124, 87.588, 15.339]
  MoveL 231 to (-185.58, -97.07, 340.79) mm, rotated rx -20 ry -0.55 rz 0.2 deg; joints [21.007, -122.284, -87.303, -50.609, 87.868, 15.437]
  MoveL 232 to (-185.05, -84.75, 336.5) mm, rotated rx -20.23 ry -0.19 rz 0.07 deg; joints [21.414, -121.044, -89.636, -49.867, 87.488, 15.853]
  MoveL 233 to (-185.03, -74.92, 332.46) mm, rotated rx -19.87 ry 0.3 rz -0.11 deg; joints [21.959, -119.787, -92.048, -48.536, 86.799, 16.382]
  MoveL 234 to (-185.07, -68.55, 330.48) mm, rotated rx -19.39 ry 0.55 rz -0.19 deg; joints [22.317, -118.967, -93.819, -47.22, 86.353, 16.716]
  MoveL 235 to (-184.98, -63.01, 328.13) mm, rotated rx -18.94 ry 0.77 rz -0.26 deg; joints [22.644, -118.176, -95.406, -46.081, 85.937, 17.02]
  MoveL 236 to (-185, -54.67, 325.38) mm, rotated rx -18.24 ry 0.8 rz -0.26 deg; joints [23.002, -117.089, -97.778, -44.159, 85.64, 17.334]
  MoveL 237 to (-185.06, -45.17, 322.86) mm, rotated rx -18.51 ry 0.68 rz -0.23 deg; joints [23.179, -116.314, -99.356, -43.589, 85.81, 17.521]
  MoveL 238 to (-185.4, -37.33, 320.37) mm, rotated rx -18.91 ry 0.65 rz -0.22 deg; joints [23.373, -115.696, -100.468, -43.479, 85.924, 17.734]
  MoveL 239 to (-184.93, -32.22, 318.4) mm, rotated rx -19.04 ry 0.64 rz -0.22 deg; joints [23.47, -115.2, -101.343, -43.233, 85.95, 17.837]
  MoveL 240 to (-185.11, -25, 315.73) mm, rotated rx -19.38 ry 0.59 rz -0.21 deg; joints [23.638, -114.575, -102.406, -43.108, 86.078, 18.02]
  MoveL 241 to (-185.24, -16.11, 311.83) mm, rotated rx -19 ry 0.89 rz -0.31 deg; joints [24.177, -113.477, -104.448, -41.946, 85.561, 18.539]
  MoveL 242 to (-186.73, -8.78, 310) mm, rotated rx -19.04 ry 0.7 rz -0.24 deg; joints [24.446, -112.88, -105.749, -41.233, 85.723, 18.801]
  MoveL 243 to (-184.56, -3.69, 308.1) mm, rotated rx -18.89 ry 0.68 rz -0.23 deg; joints [24.431, -112.283, -106.91, -40.512, 85.696, 18.777]
  MoveL 244 to (-185.07, 5.23, 305.32) mm, rotated rx -18.11 ry 0.63 rz -0.21 deg; joints [24.91, -111.232, -109.277, -38.481, 85.4, 19.2]
  MoveL 245 to (-184.86, 14.68, 301.49) mm, rotated rx -17.97 ry 0.72 rz -0.23 deg; joints [25.323, -110.211, -111.141, -37.567, 85.193, 19.6]
  MoveL 246 to (-190.7, 18.51, 299) mm, rotated rx -18.08 ry 0.45 rz -0.15 deg; joints [25.915, -109.801, -111.66, -37.52, 85.377, 20.183]
  MoveL 247 to (-189.53, 18.51, 299) mm, rotated rx -18.07 ry 0.54 rz -0.18 deg; joints [25.848, -109.782, -111.684, -37.534, 85.298, 20.119]
  MoveL 248 to (-185.09, 25.08, 298.32) mm, rotated rx -17.97 ry 0.75 rz -0.24 deg; joints [25.761, -109.287, -112.984, -36.696, 85.08, 20.033]
  MoveL 249 to (-184.93, 35.16, 295.53) mm, rotated rx -17.44 ry 0.81 rz -0.26 deg; joints [26.287, -108.294, -115.232, -35.012, 84.728, 20.516]
  MoveL 250 to (-192.37, 35.35, 295.5) mm, rotated rx -17.33 ry 0.55 rz -0.17 deg; joints [26.943, -108.365, -115.207, -34.828, 84.817, 21.144]
  MoveL 251 to (-191.54, 43.86, 292.67) mm, rotated rx -17.87 ry 0.38 rz -0.12 deg; joints [27.006, -107.712, -116.257, -34.876, 85.169, 21.24]
  MoveL 252 to (-184.99, 45.32, 292.15) mm, rotated rx -18.2 ry 0.67 rz -0.22 deg; joints [26.476, -107.563, -116.339, -35.316, 85.101, 20.75]
  MoveL 253 to (-185.24, 52.47, 290.06) mm, rotated rx -18.77 ry 0.6 rz -0.2 deg; joints [26.641, -107.108, -117.064, -35.569, 85.336, 20.949]
  MoveL 254 to (-191.25, 53.33, 290.43) mm, rotated rx -18.74 ry 0.84 rz -0.28 deg; joints [27.452, -107.22, -117.023, -35.625, 84.951, 21.756]
  MoveL 255 to (-182.98, -253.32, 400) mm, rotated rx -18.95 ry -1.32 rz 0.45 deg; joints [17.52, -143.425, -45.961, -69.509, 89.036, 11.956]
  MoveL 256 to (-184.02, -208.91, 380.62) mm, rotated rx -21.64 ry -1.07 rz 0.42 deg; joints [18.211, -137.486, -56.768, -67.329, 89.254, 12.736]
  MoveL 257 to (-184.07, -148.48, 360.07) mm, rotated rx -20.29 ry -1.51 rz 0.56 deg; joints [19.266, -128.477, -75.269, -56.427, 89.225, 13.726]
  MoveL 258 to (-181.15, -119.21, 350) mm, rotated rx -20.1 ry -0.45 rz 0.16 deg; joints [20.146, -124.93, -82.297, -53.062, 87.934, 14.593]
  MoveL 259 to (-177.94, -118.6, 350) mm, rotated rx -20.22 ry -0.28 rz 0.1 deg; joints [19.963, -124.909, -82.32, -53.223, 87.819, 14.42]
  MoveL 260 to (-184.32, -92.19, 338.59) mm, rotated rx -20.11 ry -0.45 rz 0.16 deg; joints [21.063, -121.722, -88.271, -50.34, 87.78, 15.498]
  MoveL 261 to (-183.1, 20.14, 300) mm, rotated rx -17.96 ry 0.75 rz -0.24 deg; joints [25.37, -109.719, -112.157, -37.05, 85.144, 19.647]
  MoveL 262 to (-176.96, 20.14, 300) mm, rotated rx -17.91 ry 0.73 rz -0.24 deg; joints [24.74, -109.62, -112.348, -36.854, 85.268, 19.023]
  MoveL 263 to (-183.86, 56.86, 288.43) mm, rotated rx -18.51 ry 0.75 rz -0.25 deg; joints [26.834, -106.591, -118.08, -34.901, 85.062, 21.127]
  MoveL 264 to (-182.3, 65.25, 284.97) mm, rotated rx -17.82 ry 0.63 rz -0.2 deg; joints [27.133, -105.519, -120.238, -33.141, 84.879, 21.37]
  MoveL 265 to (-182.14, 75.16, 281.95) mm, rotated rx -18.16 ry 0.38 rz -0.13 deg; joints [27.338, -104.742, -121.657, -32.747, 85.203, 21.588]
  MoveL 266 to (-181.3, 82.53, 280.25) mm, rotated rx -17.55 ry 0.15 rz -0.05 deg; joints [27.578, -104.032, -123.487, -30.982, 85.157, 21.772]
  MoveL 267 to (-175.04, -254.27, 400) mm, rotated rx -19.17 ry -1.6 rz 0.56 deg; joints [16.841, -143.621, -45.463, -69.951, 89.505, 11.297]
  MoveL 268 to (-171.57, -251.65, 399) mm, rotated rx -19.72 ry -1.27 rz 0.46 deg; joints [16.728, -143.548, -45.437, -70.656, 89.294, 11.207]
  MoveL 269 to (-174.92, -244.96, 396.27) mm, rotated rx -20.11 ry -0.99 rz 0.36 deg; joints [17.139, -142.633, -47.135, -70.32, 89.002, 11.626]
  MoveL 270 to (-175.01, -234.92, 392.38) mm, rotated rx -20.58 ry -0.93 rz 0.35 deg; joints [17.284, -141.178, -49.917, -69.472, 89.022, 11.785]
  MoveL 271 to (-175.35, -228.64, 390) mm, rotated rx -21.89 ry -0.9 rz 0.36 deg; joints [17.311, -141.096, -49.765, -70.988, 89.265, 11.854]
  MoveL 272 to (-175.04, -223.52, 388.18) mm, rotated rx -22.79 ry -1.07 rz 0.45 deg; joints [17.231, -140.913, -49.955, -71.83, 89.641, 11.8]
  MoveL 273 to (-175.18, -215.23, 386.21) mm, rotated rx -22.55 ry -1.08 rz 0.45 deg; joints [17.378, -139.426, -53.151, -69.885, 89.58, 11.938]
  MoveL 274 to (-174.53, -207.38, 381.46) mm, rotated rx -21.66 ry -0.84 rz 0.33 deg; joints [17.641, -137.306, -57.301, -67.039, 89.101, 12.174]
  MoveL 275 to (-175.61, -202.71, 378.05) mm, rotated rx -21.25 ry -0.87 rz 0.34 deg; joints [17.832, -136.132, -59.49, -65.619, 89.016, 12.349]
  MoveL 276 to (-174.91, -195.04, 376.14) mm, rotated rx -20.84 ry -0.86 rz 0.33 deg; joints [17.945, -134.826, -62.324, -63.7, 88.892, 12.447]
  MoveL 277 to (-175.17, -184.72, 373.32) mm, rotated rx -19.49 ry -0.37 rz 0.13 deg; joints [18.462, -132.705, -67.018, -59.938, 87.994, 12.909]
  MoveL 278 to (-175.73, -177.66, 370.13) mm, rotated rx -19.26 ry 0.04 rz -0.02 deg; joints [18.835, -131.581, -69.192, -58.781, 87.45, 13.271]
  MoveL 279 to (-174.65, -173.18, 368.28) mm, rotated rx -19.58 ry 0.31 rz -0.11 deg; joints [18.924, -131.131, -69.945, -58.857, 87.232, 13.374]
  MoveL 280 to (-175.15, -164.6, 365.9) mm, rotated rx -20.48 ry 0.2 rz -0.07 deg; joints [18.986, -130.573, -70.932, -59.276, 87.546, 13.47]
  MoveL 281 to (-175.06, -154.68, 362.48) mm, rotated rx -20.16 ry -0.17 rz 0.06 deg; joints [19.042, -129.14, -73.901, -57.341, 87.845, 13.51]
  MoveL 282 to (-175.03, -148.96, 360) mm, rotated rx -19.94 ry -0.38 rz 0.14 deg; joints [19.088, -128.264, -75.638, -56.219, 88.002, 13.544]
  MoveL 283 to (-175.16, -143.66, 357.95) mm, rotated rx -20.08 ry -0.51 rz 0.19 deg; joints [19.134, -127.662, -76.771, -55.79, 88.161, 13.594]
  MoveL 284 to (-174.99, -135.02, 354.93) mm, rotated rx -20.52 ry -0.79 rz 0.29 deg; joints [19.127, -126.831, -78.324, -55.43, 88.554, 13.602]
  MoveL 285 to (-175.62, -125.71, 351.58) mm, rotated rx -20.44 ry -0.47 rz 0.18 deg; joints [19.519, -125.698, -80.551, -54.349, 88.149, 13.988]
  MoveL 286 to (-171.42, -121.42, 349) mm, rotated rx -20.59 ry 0.04 rz -0.01 deg; joints [19.499, -125.113, -81.435, -54.328, 87.658, 13.98]
  MoveL 287 to (-174.43, -114.14, 347.5) mm, rotated rx -20.25 ry 0.1 rz -0.04 deg; joints [19.957, -124.275, -83.365, -52.941, 87.435, 14.419]
  MoveL 288 to (-175.06, -104.34, 343.1) mm, rotated rx -19.98 ry 0.35 rz -0.13 deg; joints [20.387, -122.952, -85.86, -51.59, 87.04, 14.835]
  MoveL 289 to (-175.03, -97.19, 340.3) mm, rotated rx -19.93 ry 0.56 rz -0.2 deg; joints [20.66, -122.111, -87.458, -50.859, 86.768, 15.105]
  MoveL 290 to (-174.95, -92.26, 338.59) mm, rotated rx -20.12 ry 0.63 rz -0.23 deg; joints [20.784, -121.65, -88.302, -50.683, 86.721, 15.238]
  MoveL 291 to (-175.02, -84.62, 335.98) mm, rotated rx -20.47 ry 0.6 rz -0.22 deg; joints [20.917, -120.973, -89.539, -50.464, 86.826, 15.384]
  MoveL 292 to (-174.8, -74.94, 332.05) mm, rotated rx -20.12 ry 0.47 rz -0.17 deg; joints [21.128, -119.717, -91.993, -48.903, 86.835, 15.575]
  MoveL 293 to (-174.94, -68.51, 330.5) mm, rotated rx -19.73 ry 0.39 rz -0.14 deg; joints [21.309, -118.966, -93.708, -47.552, 86.781, 15.735]
  MoveL 294 to (-175.21, -63.33, 327.95) mm, rotated rx -19.35 ry 0.46 rz -0.16 deg; joints [21.565, -118.19, -95.19, -46.507, 86.56, 15.97]
  MoveL 295 to (-174.68, -55.53, 325.6) mm, rotated rx -18.32 ry 0.57 rz -0.19 deg; joints [21.923, -117.057, -97.787, -44.115, 86.096, 16.271]
  MoveL 296 to (-175.01, -44.86, 322.49) mm, rotated rx -18.57 ry 0.92 rz -0.31 deg; joints [22.393, -116.146, -99.568, -43.614, 85.724, 16.755]
  MoveL 297 to (-175.76, -37.52, 320.22) mm, rotated rx -18.99 ry 1 rz -0.34 deg; joints [22.653, -115.601, -100.528, -43.653, 85.718, 17.037]
  MoveL 298 to (-174.88, -32.53, 318.34) mm, rotated rx -19.13 ry 1.08 rz -0.38 deg; joints [22.746, -115.12, -101.373, -43.452, 85.658, 17.137]
  MoveL 299 to (-174.98, -24.91, 315.43) mm, rotated rx -19.39 ry 1.11 rz -0.39 deg; joints [22.97, -114.419, -102.577, -43.229, 85.665, 17.373]
  MoveL 300 to (-174.98, -15.69, 311.69) mm, rotated rx -18.98 ry 0.97 rz -0.33 deg; joints [23.256, -113.294, -104.772, -41.743, 85.64, 17.63]
  MoveL 301 to (-172.07, -8.73, 310) mm, rotated rx -18.85 ry 1.02 rz -0.35 deg; joints [23.239, -112.627, -106.234, -40.833, 85.552, 17.607]
  MoveL 302 to (-175.48, -4.58, 308.06) mm, rotated rx -18.89 ry 0.84 rz -0.29 deg; joints [23.609, -112.208, -106.937, -40.559, 85.683, 17.97]
  MoveL 303 to (-175.18, 5.37, 305.54) mm, rotated rx -18.06 ry 0.78 rz -0.26 deg; joints [24.016, -111.11, -109.545, -38.269, 85.408, 18.32]
  MoveL 304 to (-175.17, 14.66, 302.07) mm, rotated rx -17.96 ry 0.72 rz -0.23 deg; joints [24.333, -110.156, -111.349, -37.324, 85.38, 18.624]
  MoveL 305 to (-174.98, 25.44, 298.58) mm, rotated rx -17.9 ry 0.7 rz -0.22 deg; joints [24.707, -109.147, -113.338, -36.316, 85.311, 18.989]
  MoveL 306 to (-175.18, 35.26, 295.56) mm, rotated rx -17.66 ry 0.79 rz -0.25 deg; joints [25.202, -108.213, -115.28, -35.149, 85.045, 19.462]
  MoveL 307 to (-175.05, 45.59, 291.78) mm, rotated rx -18.34 ry 0.88 rz -0.29 deg; joints [25.529, -107.396, -116.475, -35.477, 85.115, 19.832]
  MoveL 308 to (-175.12, 52.29, 290) mm, rotated rx -18.51 ry 0.94 rz -0.31 deg; joints [25.804, -106.893, -117.467, -35.193, 85.064, 20.116]
  MoveL 309 to (-174.85, 57.24, 288.4) mm, rotated rx -18.2 ry 0.82 rz -0.27 deg; joints [25.978, -106.356, -118.636, -34.236, 85.04, 20.264]
  MoveL 310 to (-175, 65.14, 285.1) mm, rotated rx -17.73 ry 0.84 rz -0.27 deg; joints [26.462, -105.418, -120.434, -32.987, 84.773, 20.709]
  MoveL 311 to (-174.94, 74.95, 281.88) mm, rotated rx -17.96 ry 0.49 rz -0.16 deg; joints [26.627, -104.586, -121.957, -32.399, 85.166, 20.877]
  MoveL 312 to (-174.86, 82.63, 280.12) mm, rotated rx -17.42 ry 0.35 rz -0.11 deg; joints [26.996, -103.884, -123.742, -30.783, 85.035, 21.197]
  MoveL 313 to (-173.26, 87.91, 278.19) mm, rotated rx -17.18 ry 0.08 rz -0.02 deg; joints [26.946, -103.308, -124.923, -29.848, 85.226, 21.12]
  MoveL 314 to (-173.49, 95.78, 275.16) mm, rotated rx -17.51 ry -0.38 rz 0.12 deg; joints [26.984, -102.613, -126.028, -29.577, 85.783, 21.169]
  MoveL 315 to (-173.08, 104.51, 272.8) mm, rotated rx -17.73 ry -0.41 rz 0.13 deg; joints [27.28, -101.959, -127.301, -29.167, 85.835, 21.475]
  MoveL 316 to (-171, 111.91, 270.57) mm, rotated rx -17.69 ry -0.68 rz 0.22 deg; joints [27.221, -101.303, -128.64, -28.344, 86.097, 21.408]
  MoveL 317 to (-171.35, 117.73, 268) mm, rotated rx -17.56 ry -1.21 rz 0.38 deg; joints [27.247, -100.666, -129.804, -27.489, 86.563, 21.409]
  MoveL 318 to (-163.89, -256.9, 400.42) mm, rotated rx -20.27 ry -0.45 rz 0.17 deg; joints [16.409, -144.964, -42.303, -73.081, 88.601, 10.915]
  MoveL 319 to (-165.63, -252.06, 399) mm, rotated rx -20.33 ry -0.8 rz 0.3 deg; joints [16.453, -144.092, -44.124, -72.119, 88.975, 10.958]
  MoveL 320 to (-165.14, -245.05, 396.86) mm, rotated rx -20.81 ry -0.64 rz 0.24 deg; joints [16.546, -143.207, -45.851, -71.788, 88.879, 11.065]
  MoveL 321 to (-164.89, -235.56, 393.03) mm, rotated rx -20.97 ry 0 rz 0 deg; joints [16.905, -141.569, -49.032, -70.543, 88.189, 11.428]
  MoveL 322 to (-163.11, -228.64, 390) mm, rotated rx -21.69 ry 0.02 rz -0.01 deg; joints [16.843, -140.835, -50.265, -70.749, 88.318, 11.389]
  MoveL 323 to (-165.49, -223.67, 387.49) mm, rotated rx -22.42 ry -0.37 rz 0.15 deg; joints [16.879, -140.475, -50.747, -71.266, 88.865, 11.443]
  MoveL 324 to (-164.76, -214.67, 385.19) mm, rotated rx -22.53 ry -0.6 rz 0.25 deg; joints [16.856, -139.122, -53.597, -69.819, 89.132, 11.422]
  MoveL 325 to (-165.05, -206.81, 381.95) mm, rotated rx -21.78 ry -0.49 rz 0.2 deg; joints [17.099, -137.29, -57.371, -67.175, 88.84, 11.642]
  MoveL 326 to (-165.4, -202.33, 378.9) mm, rotated rx -21.27 ry -0.39 rz 0.15 deg; joints [17.288, -136.102, -59.647, -65.608, 88.601, 11.815]
  MoveL 327 to (-165.18, -195.64, 375.95) mm, rotated rx -21.06 ry -0.23 rz 0.09 deg; joints [17.467, -134.92, -61.965, -64.309, 88.363, 11.986]
  MoveL 328 to (-165.01, -185.43, 373.18) mm, rotated rx -20.32 ry 0.24 rz -0.09 deg; joints [17.877, -133.142, -65.813, -61.639, 87.65, 12.37]
  MoveL 329 to (-164.28, -177.81, 370.53) mm, rotated rx -19.91 ry 0.76 rz -0.27 deg; joints [18.212, -131.893, -68.395, -60.041, 86.964, 12.691]
  MoveL 330 to (-165.33, -173, 368) mm, rotated rx -19.9 ry 0.96 rz -0.35 deg; joints [18.473, -131.178, -69.683, -59.521, 86.706, 12.951]
  MoveL 331 to (-165.29, -164.75, 364.78) mm, rotated rx -20.26 ry 1.19 rz -0.44 deg; joints [18.69, -130.269, -71.339, -59.185, 86.516, 13.181]
  MoveL 332 to (-164.95, -155.03, 362.64) mm, rotated rx -19.75 ry 1.08 rz -0.39 deg; joints [18.838, -128.914, -74.384, -56.984, 86.493, 13.307]
  MoveL 333 to (-164.56, -148.51, 360.53) mm, rotated rx -19.59 ry 0.83 rz -0.3 deg; joints [18.84, -128.038, -76.211, -55.812, 86.71, 13.299]
  MoveL 334 to (-165.14, -143.85, 357.64) mm, rotated rx -19.6 ry 0.46 rz -0.16 deg; joints [18.824, -127.332, -77.419, -55.232, 87.099, 13.278]
  MoveL 335 to (-164.74, -135.44, 354.26) mm, rotated rx -20.14 ry -0.02 rz 0.01 deg; joints [18.694, -126.522, -78.826, -55.045, 87.742, 13.167]
  MoveL 336 to (-164.65, -127.05, 351.44) mm, rotated rx -21.02 ry -0.05 rz 0.02 deg; joints [18.75, -125.958, -79.729, -55.555, 87.967, 13.254]
  MoveL 337 to (-164.92, -121.55, 348.42) mm, rotated rx -20.85 ry 0.05 rz -0.02 deg; joints [18.955, -125.109, -81.255, -54.739, 87.795, 13.451]
  MoveL 338 to (-159.19, -120.69, 349) mm, rotated rx -20.94 ry -0.07 rz 0.03 deg; joints [18.435, -125.101, -81.394, -54.654, 88.023, 12.94]
  MoveL 339 to (-164.94, -114.97, 346.4) mm, rotated rx -20.53 ry 0.28 rz -0.1 deg; joints [19.231, -124.239, -83.087, -53.536, 87.435, 13.715]
  MoveL 340 to (-164.82, -104.74, 342.69) mm, rotated rx -20.43 ry 0.65 rz -0.24 deg; joints [19.626, -123.028, -85.445, -52.408, 86.963, 14.106]
  MoveL 341 to (-164.39, -96.59, 340.41) mm, rotated rx -20.24 ry 0.83 rz -0.31 deg; joints [19.872, -122.104, -87.401, -51.25, 86.692, 14.344]
  MoveL 342 to (-165.63, -91.88, 338.77) mm, rotated rx -20.17 ry 0.96 rz -0.35 deg; joints [20.154, -121.575, -88.452, -50.713, 86.495, 14.623]
  MoveL 343 to (-165.17, -84.6, 336.41) mm, rotated rx -20.11 ry 0.68 rz -0.25 deg; joints [20.154, -120.768, -90.096, -49.743, 86.772, 14.616]
  MoveL 344 to (-164.94, -75.03, 332.3) mm, rotated rx -19.84 ry 0.36 rz -0.13 deg; joints [20.25, -119.532, -92.462, -48.272, 87.013, 14.694]
  MoveL 345 to (-165.25, -68.9, 330) mm, rotated rx -19.58 ry 0.33 rz -0.12 deg; joints [20.443, -118.765, -94.009, -47.238, 86.952, 14.872]
  MoveL 346 to (-164.64, -64.28, 327.76) mm, rotated rx -19.25 ry 0.17 rz -0.06 deg; joints [20.477, -118.071, -95.352, -46.229, 87.017, 14.889]
  MoveL 347 to (-164.78, -55.37, 324.52) mm, rotated rx -18.8 ry 0.28 rz -0.09 deg; joints [20.829, -116.969, -97.6, -44.691, 86.733, 15.214]
  MoveL 348 to (-165, -44.72, 321.63) mm, rotated rx -18.98 ry 0.87 rz -0.3 deg; joints [21.406, -116.062, -99.408, -44.178, 86.066, 15.803]
  MoveL 349 to (-163.95, -38.25, 320.06) mm, rotated rx -19.29 ry 1.24 rz -0.43 deg; joints [21.628, -115.595, -100.318, -44.148, 85.736, 16.045]
  MoveL 350 to (-165.45, -33.46, 318.13) mm, rotated rx -19.25 ry 1.31 rz -0.46 deg; joints [21.952, -115.084, -101.258, -43.729, 85.594, 16.364]
  MoveL 351 to (-164.92, -25.17, 314.83) mm, rotated rx -19.26 ry 1.23 rz -0.43 deg; joints [22.104, -114.196, -102.879, -42.991, 85.658, 16.514]
  MoveL 352 to (-165.04, -15.67, 311.4) mm, rotated rx -18.98 ry 1.22 rz -0.42 deg; joints [22.443, -113.14, -104.967, -41.707, 85.527, 16.833]
  MoveL 353 to (-165.39, -8.84, 310) mm, rotated rx -18.68 ry 1.17 rz -0.4 deg; joints [22.693, -112.504, -106.497, -40.533, 85.45, 17.063]
  MoveL 354 to (-164.64, -3.21, 307.73) mm, rotated rx -18.36 ry 0.87 rz -0.29 deg; joints [22.691, -111.801, -107.908, -39.429, 85.658, 17.036]
  MoveL 355 to (-165.14, 5.34, 304.94) mm, rotated rx -17.98 ry 0.48 rz -0.16 deg; joints [22.86, -110.887, -109.869, -37.912, 85.911, 17.171]
  MoveL 356 to (-165.02, 14.69, 301.2) mm, rotated rx -17.92 ry 0.35 rz -0.11 deg; joints [23.105, -109.902, -111.665, -37.016, 85.978, 17.406]
  MoveL 357 to (-164.13, 18.51, 299) mm, rotated rx -18.01 ry 0.33 rz -0.11 deg; joints [23.132, -109.431, -112.319, -36.917, 86.021, 17.437]
  MoveL 358 to (-164.93, 24.59, 298.14) mm, rotated rx -17.98 ry 0.37 rz -0.12 deg; joints [23.437, -109.025, -113.377, -36.272, 85.911, 17.736]
  MoveL 359 to (-164.92, 35.23, 295.33) mm, rotated rx -17.94 ry 0.62 rz -0.2 deg; joints [23.967, -108.129, -115.26, -35.361, 85.538, 18.261]
  MoveL 360 to (-164.93, 45.4, 291.66) mm, rotated rx -18.3 ry 0.89 rz -0.29 deg; joints [24.448, -107.247, -116.7, -35.273, 85.296, 18.764]
  MoveL 361 to (-166.06, 51.62, 290) mm, rotated rx -18.48 ry 0.99 rz -0.33 deg; joints [24.833, -106.795, -117.58, -35.078, 85.182, 19.158]
  MoveL 362 to (-164.84, 56.36, 288.17) mm, rotated rx -18.12 ry 0.74 rz -0.24 deg; joints [24.81, -106.213, -118.788, -34.031, 85.323, 19.106]
  MoveL 363 to (-165.09, 65.22, 284.77) mm, rotated rx -17.71 ry 0.77 rz -0.25 deg; joints [25.321, -105.232, -120.697, -32.769, 85.053, 19.582]
  MoveL 364 to (-165.02, 75, 282.24) mm, rotated rx -17.65 ry 0.48 rz -0.15 deg; joints [25.547, -104.435, -122.446, -31.669, 85.278, 19.792]
  MoveL 365 to (-165.06, 82.54, 280.38) mm, rotated rx -17.23 ry 0.27 rz -0.09 deg; joints [25.835, -103.762, -124.102, -30.244, 85.28, 20.039]
  MoveL 366 to (-164.95, 87.76, 278.44) mm, rotated rx -17.14 ry -0.01 rz 0 deg; joints [25.902, -103.241, -125.112, -29.568, 85.51, 20.09]
  MoveL 367 to (-164.89, 94.75, 275.69) mm, rotated rx -17.24 ry -0.06 rz 0.02 deg; joints [26.172, -102.564, -126.221, -29.238, 85.543, 20.361]
  MoveL 368 to (-164.87, 104.55, 273.24) mm, rotated rx -17.6 ry -0.05 rz 0.02 deg; joints [26.542, -101.892, -127.522, -28.981, 85.586, 20.751]
  MoveL 369 to (-164.1, 111.59, 270.32) mm, rotated rx -17.35 ry -0.28 rz 0.09 deg; joints [26.715, -101.102, -128.978, -28.006, 85.688, 20.896]
  MoveL 370 to (-165.22, 116.75, 268.64) mm, rotated rx -17.3 ry -0.6 rz 0.19 deg; joints [26.91, -100.655, -129.896, -27.381, 85.942, 21.074]
  MoveL 371 to (-165.65, 120.38, 268.29) mm, rotated rx -17.34 ry -0.89 rz 0.28 deg; joints [26.923, -100.503, -130.469, -26.886, 86.227, 21.083]
  MoveL 372 to (-162.68, 121.15, 270) mm, rotated rx -17.24 ry -0.67 rz 0.21 deg; joints [26.714, -100.72, -130.65, -26.463, 86.022, 20.875]
  MoveL 373 to (-155.36, -254.91, 401.11) mm, rotated rx -19.69 ry 0.36 rz -0.13 deg; joints [16.198, -144.151, -44.253, -71.531, 87.68, 10.693]
  MoveL 374 to (-155.09, -244.95, 396.46) mm, rotated rx -20.98 ry -0.19 rz 0.07 deg; joints [16.021, -143.195, -45.748, -72.143, 88.525, 10.555]
  MoveL 375 to (-154.67, -235.1, 392.45) mm, rotated rx -21.24 ry -0.12 rz 0.05 deg; joints [16.14, -141.54, -48.96, -70.862, 88.48, 10.68]
  MoveL 376 to (-154.54, -228.69, 390.67) mm, rotated rx -21.61 ry 0.06 rz -0.02 deg; joints [16.262, -140.767, -50.505, -70.489, 88.345, 10.811]
  MoveL 377 to (-155.4, -223.11, 387.7) mm, rotated rx -22.19 ry 0.06 rz -0.03 deg; joints [16.369, -140.155, -51.468, -70.715, 88.432, 10.933]
  MoveL 378 to (-155.02, -214.61, 384.8) mm, rotated rx -22.47 ry -0.06 rz 0.02 deg; joints [16.394, -138.949, -53.861, -69.776, 88.611, 10.964]
  MoveL 379 to (-154.99, -206.21, 381.5) mm, rotated rx -21.87 ry 0.08 rz -0.03 deg; joints [16.617, -137.155, -57.542, -67.341, 88.321, 11.171]
  MoveL 380 to (-155.21, -202.38, 379) mm, rotated rx -21.38 ry 0.07 rz -0.03 deg; joints [16.734, -136.115, -59.568, -65.877, 88.214, 11.273]
  MoveL 381 to (-154.72, -195.38, 376.25) mm, rotated rx -21.18 ry 0.01 rz 0 deg; joints [16.797, -134.91, -61.992, -64.441, 88.232, 11.328]
  MoveL 382 to (-155.24, -185.27, 373.18) mm, rotated rx -21.14 ry 0.18 rz -0.07 deg; joints [17.063, -133.516, -64.86, -62.977, 88.01, 11.591]
  MoveL 383 to (-155.59, -177.09, 370.84) mm, rotated rx -20.35 ry 0.8 rz -0.3 deg; joints [17.545, -132.022, -68.1, -60.61, 87.127, 12.048]
  MoveL 384 to (-154.53, -172.3, 368.33) mm, rotated rx -20.28 ry 1 rz -0.37 deg; joints [17.647, -131.253, -69.513, -59.949, 86.883, 12.149]
  MoveL 385 to (-155.09, -164.93, 364.23) mm, rotated rx -20.3 ry 1.08 rz -0.4 deg; joints [17.865, -130.142, -71.474, -59.148, 86.765, 12.366]
  MoveL 386 to (-154.97, -155.24, 361.48) mm, rotated rx -19.77 ry 1.03 rz -0.37 deg; joints [18.045, -128.714, -74.561, -56.968, 86.686, 12.524]
  MoveL 387 to (-157.62, -148.29, 360.2) mm, rotated rx -19.08 ry 1.04 rz -0.36 deg; joints [18.442, -127.679, -77.007, -54.91, 86.451, 12.889]
  MoveL 388 to (-154.26, -143.59, 357.88) mm, rotated rx -18.82 ry 0.63 rz -0.21 deg; joints [18.112, -126.88, -78.57, -53.779, 86.882, 12.548]
  MoveL 389 to (-155.18, -135.02, 355.02) mm, rotated rx -19.83 ry 0.28 rz -0.1 deg; joints [18.093, -126.349, -79.377, -54.407, 87.467, 12.565]
  MoveL 390 to (-154.86, -125.16, 351.56) mm, rotated rx -20.89 ry -0.13 rz 0.05 deg; joints [17.968, -125.676, -80.445, -54.946, 88.144, 12.476]
  MoveL 391 to (-153.7, -119.21, 350) mm, rotated rx -20.93 ry -0.23 rz 0.09 deg; joints [17.931, -125.052, -81.758, -54.274, 88.265, 12.44]
  MoveL 392 to (-155.18, -114.52, 347.23) mm, rotated rx -20.98 ry -0.08 rz 0.03 deg; joints [18.219, -124.415, -82.799, -53.959, 88.069, 12.727]
  MoveL 393 to (-155, -104.66, 342.53) mm, rotated rx -20.55 ry 0.26 rz -0.1 deg; joints [18.617, -122.96, -85.533, -52.358, 87.554, 13.108]
  MoveL 394 to (-155.42, -96.62, 340.35) mm, rotated rx -19.99 ry 0.08 rz -0.03 deg; joints [18.786, -121.901, -87.889, -50.484, 87.585, 13.252]
  MoveL 395 to (-154.61, -91.88, 338.44) mm, rotated rx -19.73 ry -0.19 rz 0.07 deg; joints [18.714, -121.234, -89.246, -49.464, 87.825, 13.168]
  MoveL 396 to (-155.18, -84.54, 336.31) mm, rotated rx -19.8 ry -0.42 rz 0.15 deg; joints [18.797, -120.522, -90.716, -48.722, 88.064, 13.251]
  MoveL 397 to (-155.09, -74.97, 332.55) mm, rotated rx -20.1 ry -0.42 rz 0.15 deg; joints [18.972, -119.569, -92.405, -48.292, 88.098, 13.436]
  MoveL 398 to (-154.19, -68.71, 330.37) mm, rotated rx -19.83 ry -0.18 rz 0.06 deg; joints [19.183, -118.792, -93.982, -47.289, 87.751, 13.635]
  MoveL 399 to (-155.11, -63.42, 328.04) mm, rotated rx -19.26 ry 0.12 rz -0.04 deg; joints [19.61, -117.971, -95.641, -45.992, 87.23, 14.034]
  MoveL 400 to (-155.2, -54.9, 325.17) mm, rotated rx -19.16 ry 0.49 rz -0.17 deg; joints [20.024, -117.069, -97.414, -45.145, 86.75, 14.443]
  MoveL 401 to (-155.03, -44.89, 321.74) mm, rotated rx -19.5 ry 0.66 rz -0.23 deg; joints [20.305, -116.172, -99.036, -44.809, 86.612, 14.738]
  MoveL 402 to (-156.35, -38.19, 320.13) mm, rotated rx -19.55 ry 0.93 rz -0.33 deg; joints [20.726, -115.615, -100.219, -44.332, 86.277, 15.16]
  MoveL 403 to (-154.41, -34.09, 317.83) mm, rotated rx -19.38 ry 0.67 rz -0.24 deg; joints [20.553, -115.01, -101.28, -43.629, 86.526, 14.977]
  MoveL 404 to (-155.03, -25.67, 314.33) mm, rotated rx -19.12 ry 0.88 rz -0.31 deg; joints [20.994, -114.01, -103.152, -42.593, 86.169, 15.403]
  MoveL 405 to (-155.03, -15.79, 311.35) mm, rotated rx -19.05 ry 1.09 rz -0.38 deg; joints [21.391, -113.064, -105.064, -41.642, 85.865, 15.796]
  MoveL 406 to (-155.63, -9.8, 310) mm, rotated rx -18.45 ry 1 rz -0.33 deg; joints [21.653, -112.382, -106.741, -40.063, 85.748, 16.022]
  MoveL 407 to (-154.89, -4.48, 307.96) mm, rotated rx -17.86 ry 0.75 rz -0.24 deg; joints [21.692, -111.65, -108.338, -38.56, 85.834, 16.023]
  MoveL 408 to (-154.81, 5.33, 303.57) mm, rotated rx -17.8 ry 0.46 rz -0.15 deg; joints [21.85, -110.548, -110.267, -37.598, 86.077, 16.168]
  MoveL 409 to (-154.99, 14.66, 301.38) mm, rotated rx -17.87 ry 0.45 rz -0.14 deg; joints [22.13, -109.816, -111.861, -36.818, 86.058, 16.447]
  MoveL 410 to (-154.13, 20.85, 300) mm, rotated rx -17.9 ry 0.29 rz -0.09 deg; joints [22.136, -109.336, -112.942, -36.207, 86.221, 16.452]
  MoveL 411 to (-155.42, 25.81, 298.09) mm, rotated rx -17.91 ry 0.2 rz -0.06 deg; joints [22.383, -108.851, -113.823, -35.806, 86.272, 16.693]
  MoveL 412 to (-154.89, 35.19, 294.81) mm, rotated rx -18.28 ry 0.07 rz -0.02 deg; joints [22.507, -108.055, -115.176, -35.574, 86.485, 16.833]
  MoveL 413 to (-155, 45.44, 291.39) mm, rotated rx -18.61 ry 0.33 rz -0.11 deg; joints [22.982, -107.192, -116.659, -35.381, 86.222, 17.325]
  MoveL 414 to (-157.67, 51.3, 290) mm, rotated rx -18.35 ry 0.66 rz -0.22 deg; joints [23.729, -106.684, -117.83, -34.628, 85.673, 18.053]
  MoveL 415 to (-155.04, 55.84, 288.22) mm, rotated rx -18 ry 0.39 rz -0.13 deg; joints [23.512, -106.111, -119.024, -33.563, 85.878, 17.811]
  MoveL 416 to (-154.98, 65.44, 284.89) mm, rotated rx -17.73 ry 0.47 rz -0.15 deg; joints [23.979, -105.141, -120.927, -32.433, 85.629, 18.255]
  MoveL 417 to (-154.93, 75.06, 282.33) mm, rotated rx -17.36 ry 0.49 rz -0.15 deg; joints [24.442, -104.274, -122.887, -31.031, 85.399, 18.687]
  MoveL 418 to (-155.1, 81.83, 280.33) mm, rotated rx -17.06 ry 0.36 rz -0.11 deg; joints [24.724, -103.636, -124.313, -29.933, 85.371, 18.939]
  MoveL 419 to (-154.71, 86.98, 278) mm, rotated rx -16.99 ry 0.28 rz -0.09 deg; joints [24.88, -103.052, -125.283, -29.466, 85.391, 19.084]
  MoveL 420 to (-154.87, 94.63, 275.87) mm, rotated rx -17.22 ry 0.05 rz -0.02 deg; joints [25.025, -102.485, -126.375, -29.099, 85.665, 19.237]
  MoveL 421 to (-154.85, 104.77, 273.06) mm, rotated rx -17.37 ry -0.01 rz 0 deg; joints [25.402, -101.695, -127.939, -28.47, 85.695, 19.616]
  MoveL 422 to (-154.58, 112.24, 270.52) mm, rotated rx -16.75 ry -0.47 rz 0.14 deg; joints [25.552, -100.905, -129.781, -26.682, 85.908, 19.706]
  MoveL 423 to (-155.81, 116.64, 268.56) mm, rotated rx -16.81 ry -0.77 rz 0.23 deg; joints [25.706, -100.459, -130.487, -26.38, 86.194, 19.853]
  MoveL 424 to (-155.04, 120.7, 269) mm, rotated rx -17.12 ry -0.8 rz 0.25 deg; joints [25.67, -100.464, -130.851, -26.295, 86.332, 19.841]
  MoveL 425 to (-146.67, -255.12, 400.2) mm, rotated rx -18.33 ry 0.42 rz -0.14 deg; joints [15.719, -142.846, -47.098, -68.64, 87.465, 10.175]
  MoveL 426 to (-143.18, -252, 399) mm, rotated rx -18.38 ry 0.07 rz -0.02 deg; joints [15.382, -142.272, -48.248, -68.043, 87.9, 9.843]
  MoveL 427 to (-145.09, -244.88, 396.37) mm, rotated rx -20.42 ry -0.27 rz 0.1 deg; joints [15.341, -142.609, -47.05, -70.843, 88.617, 9.866]
  MoveL 428 to (-144.92, -235.65, 393.17) mm, rotated rx -21.39 ry -0.39 rz 0.15 deg; joints [15.338, -141.732, -48.619, -71.088, 88.907, 9.889]
  MoveL 429 to (-144.69, -228.99, 390.91) mm, rotated rx -21.79 ry -0.34 rz 0.14 deg; joints [15.398, -140.884, -50.258, -70.699, 88.922, 9.959]
  MoveL 430 to (-144.96, -223.3, 387.79) mm, rotated rx -22.24 ry -0.3 rz 0.12 deg; joints [15.484, -140.128, -51.521, -70.643, 88.948, 10.055]
  MoveL 431 to (-145.09, -214.8, 384.03) mm, rotated rx -22.49 ry -0.3 rz 0.12 deg; joints [15.595, -138.814, -54.004, -69.725, 88.974, 10.172]
  MoveL 432 to (-145.06, -206.91, 381.32) mm, rotated rx -22.12 ry -0.2 rz 0.08 deg; joints [15.764, -137.301, -57.133, -67.768, 88.786, 10.33]
  MoveL 433 to (-144.55, -201.59, 379) mm, rotated rx -21.35 ry -0.09 rz 0.04 deg; joints [15.904, -135.916, -60.015, -65.532, 88.508, 10.449]
  MoveL 434 to (-145.09, -195.15, 376.77) mm, rotated rx -21.02 ry 0.03 rz -0.01 deg; joints [16.109, -134.776, -62.378, -64.021, 88.289, 10.644]
  MoveL 435 to (-144.72, -184.59, 372.75) mm, rotated rx -21.31 ry -0.3 rz 0.12 deg; joints [16.078, -133.415, -65.006, -62.971, 88.697, 10.62]
  MoveL 436 to (-144.69, -177.81, 370.53) mm, rotated rx -21 ry -0.36 rz 0.14 deg; joints [16.177, -132.319, -67.299, -61.458, 88.677, 10.708]
  MoveL 437 to (-145.01, -172.87, 367.8) mm, rotated rx -20.66 ry -0.06 rz 0.02 deg; joints [16.438, -131.36, -69.125, -60.323, 88.257, 10.957]
  MoveL 438 to (-145.06, -165.17, 364.52) mm, rotated rx -20.29 ry 0.29 rz -0.11 deg; joints [16.748, -130.096, -71.625, -58.807, 87.773, 11.254]
  MoveL 439 to (-145.24, -155.37, 361.18) mm, rotated rx -19.76 ry 0.17 rz -0.06 deg; joints [16.911, -128.598, -74.766, -56.63, 87.77, 11.396]
  MoveL 440 to (-140.77, -150.42, 359) mm, rotated rx -19.06 ry -0.11 rz 0.04 deg; joints [16.579, -127.569, -76.947, -54.716, 87.984, 11.042]
  MoveL 441 to (-145.12, -144.15, 357.67) mm, rotated rx -18.55 ry 0.09 rz -0.03 deg; joints [17.159, -126.704, -78.953, -53.14, 87.563, 11.593]
  MoveL 442 to (-145, -134.65, 354.69) mm, rotated rx -19.47 ry -0.03 rz 0.01 deg; joints [17.176, -126.043, -80.057, -53.579, 87.873, 11.645]
  MoveL 443 to (-144.91, -125.35, 351.55) mm, rotated rx -20.56 ry -0.45 rz 0.17 deg; joints [17.043, -125.469, -80.934, -54.25, 88.555, 11.549]
  MoveL 444 to (-148.22, -119.21, 350) mm, rotated rx -20.95 ry -0.52 rz 0.2 deg; joints [17.35, -125.023, -81.823, -54.179, 88.657, 11.865]
  MoveL 445 to (-144.47, -115.01, 346.73) mm, rotated rx -21.35 ry -0.33 rz 0.13 deg; joints [17.186, -124.496, -82.426, -54.534, 88.565, 11.716]
  MoveL 446 to (-145.06, -105.15, 343.25) mm, rotated rx -20.56 ry -0.4 rz 0.15 deg; joints [17.458, -123.013, -85.551, -52.11, 88.431, 11.959]
  MoveL 447 to (-144.89, -97.16, 340.44) mm, rotated rx -19.89 ry -0.31 rz 0.11 deg; joints [17.701, -121.832, -88.052, -50.153, 88.162, 12.175]
  MoveL 448 to (-145.06, -92.21, 338) mm, rotated rx -19.52 ry -0.25 rz 0.09 deg; joints [17.884, -121.058, -89.544, -49.1, 87.989, 12.342]
  MoveL 449 to (-144.6, -84.54, 334.76) mm, rotated rx -19.68 ry -0.26 rz 0.09 deg; joints [17.987, -120.222, -91.025, -48.611, 88.008, 12.45]
  MoveL 450 to (-144.83, -74.96, 332) mm, rotated rx -20.12 ry -0.43 rz 0.16 deg; joints [18.066, -119.444, -92.527, -48.284, 88.272, 12.543]
  MoveL 451 to (-144.52, -67.81, 330.45) mm, rotated rx -19.92 ry -0.63 rz 0.23 deg; joints [18.098, -118.72, -94.191, -47.099, 88.433, 12.566]
  MoveL 452 to (-145.18, -62.35, 328.05) mm, rotated rx -19.69 ry -0.46 rz 0.16 deg; joints [18.395, -118, -95.555, -46.276, 88.143, 12.85]
  MoveL 453 to (-145.03, -54.67, 325.57) mm, rotated rx -19.32 ry -0.28 rz 0.1 deg; joints [18.68, -117.092, -97.457, -44.98, 87.827, 13.118]
  MoveL 454 to (-144.91, -44.94, 321.88) mm, rotated rx -19.59 ry -0.02 rz 0.01 deg; joints [19.002, -116.149, -99.112, -44.601, 87.561, 13.448]
  MoveL 455 to (-144.29, -38.74, 320) mm, rotated rx -19.71 ry 0.14 rz -0.05 deg; joints [19.154, -115.591, -100.192, -44.242, 87.404, 13.605]
  MoveL 456 to (-145.12, -34.72, 317.87) mm, rotated rx -19.57 ry 0.16 rz -0.06 deg; joints [19.369, -115.048, -101.134, -43.725, 87.306, 13.811]
  MoveL 457 to (-145, -25.89, 314.35) mm, rotated rx -19.43 ry 0.38 rz -0.14 deg; joints [19.72, -114.054, -102.976, -42.82, 86.983, 14.154]
  MoveL 458 to (-144.98, -15.56, 311.26) mm, rotated rx -19.03 ry 0.55 rz -0.19 deg; joints [20.123, -112.954, -105.305, -41.266, 86.646, 14.535]
  MoveL 459 to (-144.56, -9.38, 310) mm, rotated rx -18.13 ry 0.39 rz -0.13 deg; joints [20.27, -112.177, -107.323, -39.115, 86.558, 14.633]
  MoveL 460 to (-145.17, -3.9, 307.93) mm, rotated rx -17.71 ry 0.38 rz -0.12 deg; joints [20.543, -111.499, -108.749, -37.97, 86.404, 14.878]
  MoveL 461 to (-145.02, 5.27, 303.87) mm, rotated rx -17.68 ry 0.25 rz -0.08 deg; joints [20.739, -110.486, -110.503, -37.182, 86.484, 15.067]
  MoveL 462 to (-145.07, 14.83, 302.15) mm, rotated rx -17.66 ry -0.17 rz 0.05 deg; joints [20.764, -109.793, -112.229, -36.017, 86.903, 15.084]
  MoveL 463 to (-144.52, 21.33, 300.45) mm, rotated rx -17.46 ry -0.45 rz 0.14 deg; joints [20.764, -109.2, -113.598, -34.967, 87.128, 15.069]
  MoveL 464 to (-145.3, 26.39, 297.75) mm, rotated rx -17.59 ry -0.57 rz 0.18 deg; joints [20.92, -108.63, -114.417, -34.821, 87.26, 15.228]
  MoveL 465 to (-145.22, 35.26, 294.93) mm, rotated rx -18.44 ry -0.46 rz 0.15 deg; joints [21.122, -108.052, -115.2, -35.478, 87.329, 15.473]
  MoveL 466 to (-145.04, 45.11, 291.25) mm, rotated rx -18.81 ry -0.13 rz 0.04 deg; joints [21.569, -107.171, -116.595, -35.439, 87.008, 15.937]
  MoveL 467 to (-142.4, 49.61, 289) mm, rotated rx -18.63 ry -0.17 rz 0.06 deg; joints [21.44, -106.575, -117.618, -34.812, 87.028, 15.8]
  MoveL 468 to (-145.04, 55.41, 287.94) mm, rotated rx -18.16 ry -0.08 rz 0.03 deg; joints [22.057, -106.059, -118.989, -33.573, 86.685, 16.382]
  MoveL 469 to (-144.96, 65.17, 284.85) mm, rotated rx -17.79 ry 0.05 rz -0.02 deg; joints [22.546, -105.086, -121.011, -32.228, 86.35, 16.842]
  MoveL 470 to (-144.87, 74.85, 281.98) mm, rotated rx -17.29 ry 0.01 rz 0 deg; joints [22.961, -104.14, -123.113, -30.61, 86.161, 17.218]
  MoveL 471 to (-144.63, 81.36, 280.19) mm, rotated rx -17.1 ry 0.08 rz -0.03 deg; joints [23.267, -103.564, -124.375, -29.791, 85.967, 17.507]
  MoveL 472 to (-144.85, 86.42, 278.11) mm, rotated rx -16.98 ry 0.24 rz -0.07 deg; joints [23.64, -103.009, -125.346, -29.328, 85.692, 17.867]
  MoveL 473 to (-145, 94.91, 275.79) mm, rotated rx -17.18 ry 0.22 rz -0.07 deg; joints [23.952, -102.366, -126.582, -28.952, 85.705, 18.187]
  MoveL 474 to (-144.91, 104.53, 273.06) mm, rotated rx -16.99 ry 0.07 rz -0.02 deg; joints [24.288, -101.539, -128.373, -27.775, 85.726, 18.499]
  MoveL 475 to (-145.78, 113.09, 270.83) mm, rotated rx -16.48 ry -0.09 rz 0.03 deg; joints [24.779, -100.792, -130.232, -26.158, 85.617, 18.939]
  MoveL 476 to (-134.59, -254.42, 398.21) mm, rotated rx -17.95 ry -0.32 rz 0.1 deg; joints [14.64, -142.118, -48.448, -67.477, 88.383, 9.1]
  MoveL 477 to (-135.07, -245.9, 396.63) mm, rotated rx -19.64 ry -0.5 rz 0.18 deg; joints [14.592, -142.083, -48.296, -69.298, 88.861, 9.104]
  MoveL 478 to (-135.27, -236.31, 394.29) mm, rotated rx -21.16 ry -0.7 rz 0.27 deg; joints [14.543, -141.704, -48.868, -70.571, 89.322, 9.097]
  MoveL 479 to (-135.18, -228.29, 391.05) mm, rotated rx -21.63 ry -0.92 rz 0.36 deg; joints [14.519, -140.624, -50.898, -70.051, 89.633, 9.084]
  MoveL 480 to (-135.09, -221.89, 387.1) mm, rotated rx -22.36 ry -0.85 rz 0.35 deg; joints [14.581, -139.893, -51.964, -70.44, 89.67, 9.162]
  MoveL 481 to (-134.97, -214.07, 383.87) mm, rotated rx -22.66 ry -0.6 rz 0.25 deg; joints [14.751, -138.77, -54.077, -69.795, 89.435, 9.337]
  MoveL 482 to (-135.02, -206.54, 381.18) mm, rotated rx -22.26 ry -0.42 rz 0.17 deg; joints [14.95, -137.276, -57.155, -67.848, 89.145, 9.526]
  MoveL 483 to (-134.17, -201.77, 379) mm, rotated rx -21.65 ry -0.29 rz 0.12 deg; joints [15.044, -136.079, -59.61, -66.02, 88.897, 9.606]
  MoveL 484 to (-135.27, -195.85, 376.55) mm, rotated rx -21.13 ry -0.28 rz 0.11 deg; joints [15.246, -134.836, -62.168, -64.2, 88.764, 9.792]
  MoveL 485 to (-134.96, -185.33, 372.5) mm, rotated rx -20.75 ry -0.53 rz 0.2 deg; joints [15.29, -133.079, -65.737, -61.97, 88.951, 9.824]
  MoveL 486 to (-135.55, -177.58, 370.29) mm, rotated rx -21 ry -0.89 rz 0.34 deg; joints [15.265, -132.228, -67.48, -61.256, 89.381, 9.805]
  MoveL 487 to (-134.61, -172.96, 368.38) mm, rotated rx -21.15 ry -1 rz 0.39 deg; joints [15.2, -131.656, -68.546, -60.886, 89.537, 9.745]
  MoveL 488 to (-135.18, -165.33, 365.12) mm, rotated rx -20.61 ry -0.76 rz 0.29 deg; joints [15.499, -130.294, -71.286, -59.025, 89.141, 10.025]
  MoveL 489 to (-134.82, -156.26, 361.1) mm, rotated rx -19.73 ry -0.55 rz 0.2 deg; joints [15.769, -128.593, -74.755, -56.435, 88.712, 10.266]
  MoveL 490 to (-135.03, -150.85, 359) mm, rotated rx -19.26 ry -0.42 rz 0.15 deg; joints [15.963, -127.677, -76.662, -55.015, 88.459, 10.442]
  MoveL 491 to (-135.13, -144.66, 357.74) mm, rotated rx -18.81 ry -0.12 rz 0.04 deg; joints [16.231, -126.821, -78.629, -53.527, 88.016, 10.691]
  MoveL 492 to (-134.87, -135.27, 354.85) mm, rotated rx -19.37 ry 0.41 rz -0.15 deg; joints [16.559, -126.007, -80.119, -53.513, 87.5, 11.037]
  MoveL 493 to (-135.18, -125.47, 352.25) mm, rotated rx -20.26 ry 0.59 rz -0.22 deg; joints [16.746, -125.37, -81.258, -53.938, 87.46, 11.254]
  MoveL 494 to (-131.48, -118.84, 350) mm, rotated rx -20.95 ry 0.76 rz -0.29 deg; joints [16.581, -124.911, -81.98, -54.38, 87.43, 11.114]
  MoveL 495 to (-134.95, -114.44, 346.74) mm, rotated rx -21.24 ry 0.2 rz -0.08 deg; joints [16.671, -124.354, -82.732, -54.357, 88.06, 11.207]
  MoveL 496 to (-135.35, -104.74, 343.05) mm, rotated rx -20.58 ry 0.1 rz -0.04 deg; joints [16.887, -122.92, -85.677, -52.187, 88.003, 11.399]
  MoveL 497 to (-135.45, -96.61, 340.38) mm, rotated rx -19.98 ry 0.1 rz -0.04 deg; joints [17.096, -121.777, -88.12, -50.305, 87.849, 11.586]
  MoveL 498 to (-134.68, -91.77, 338.52) mm, rotated rx -19.57 ry 0.14 rz -0.05 deg; joints [17.177, -121.054, -89.626, -49.127, 87.719, 11.651]
  MoveL 499 to (-135.08, -84.78, 336.87) mm, rotated rx -19.57 ry 0.13 rz -0.05 deg; joints [17.335, -120.395, -91.063, -48.356, 87.694, 11.807]
  MoveL 500 to (-134.94, -75.05, 332.62) mm, rotated rx -19.65 ry -0.03 rz 0.01 deg; joints [17.43, -119.285, -93.053, -47.522, 87.868, 11.902]
  MoveL 501 to (-136.05, -68.64, 330.06) mm, rotated rx -19.76 ry -0.38 rz 0.14 deg; joints [17.474, -118.621, -94.276, -46.997, 88.245, 11.947]
  MoveL 502 to (-134.72, -63.72, 328.22) mm, rotated rx -19.81 ry -0.37 rz 0.13 deg; joints [17.455, -118.102, -95.243, -46.6, 88.247, 11.93]
  MoveL 503 to (-134.67, -54.78, 324.84) mm, rotated rx -19.67 ry -0.11 rz 0.04 deg; joints [17.787, -117.082, -97.192, -45.602, 87.887, 12.253]
  MoveL 504 to (-134.88, -44.89, 322.31) mm, rotated rx -19.92 ry 0.14 rz -0.05 deg; joints [18.111, -116.268, -98.844, -45.079, 87.627, 12.585]
  MoveL 505 to (-130.35, -38.18, 320) mm, rotated rx -19.71 ry -0.03 rz 0.01 deg; joints [17.767, -115.495, -100.422, -44.011, 87.817, 12.236]
  MoveL 506 to (-134.98, -35.09, 317.97) mm, rotated rx -19.57 ry 0.04 rz -0.02 deg; joints [18.338, -115.028, -101.168, -43.635, 87.611, 12.793]
  MoveL 507 to (-134.93, -25.66, 314.53) mm, rotated rx -19.46 ry -0.14 rz 0.05 deg; joints [18.469, -114.024, -103.115, -42.549, 87.748, 12.916]
  MoveL 508 to (-134.99, -15.86, 311.27) mm, rotated rx -18.99 ry -0.17 rz 0.06 deg; joints [18.744, -112.912, -105.437, -40.883, 87.628, 13.167]
  MoveL 509 to (-136.79, -9.6, 310) mm, rotated rx -18.25 ry -0.04 rz 0.01 deg; joints [19.238, -112.188, -107.272, -39.107, 87.223, 13.62]
  MoveL 510 to (-134.58, -4.3, 307.53) mm, rotated rx -17.74 ry 0.05 rz -0.02 deg; joints [19.275, -111.424, -108.784, -37.887, 87.007, 13.632]
  MoveL 511 to (-135.12, 5.3, 304.07) mm, rotated rx -17.24 ry -0.15 rz 0.05 deg; joints [19.545, -110.343, -111.039, -36.189, 87.03, 13.868]
  MoveL 512 to (-135.04, 14.69, 301.97) mm, rotated rx -17.14 ry -0.59 rz 0.18 deg; joints [19.537, -109.594, -112.816, -34.951, 87.456, 13.85]
  MoveL 513 to (-135.64, 21.54, 300.38) mm, rotated rx -17.21 ry -0.79 rz 0.24 deg; joints [19.657, -109.082, -113.964, -34.336, 87.647, 13.968]
  MoveL 514 to (-134.79, 26.72, 298.12) mm, rotated rx -17.64 ry -0.77 rz 0.24 deg; joints [19.666, -108.637, -114.513, -34.662, 87.735, 14.001]
  MoveL 515 to (-135.02, 35.14, 295.08) mm, rotated rx -18.74 ry -0.54 rz 0.18 deg; joints [19.913, -108.113, -114.992, -35.843, 87.729, 14.3]
  MoveL 516 to (-135.07, 45.62, 291.9) mm, rotated rx -18.92 ry -0.52 rz 0.18 deg; joints [20.214, -107.232, -116.675, -35.231, 87.69, 14.605]
  MoveL 517 to (-131.9, 51.3, 290) mm, rotated rx -18.69 ry -0.41 rz 0.14 deg; joints [20.134, -106.624, -117.907, -34.405, 87.541, 14.517]
  MoveL 518 to (-135.14, 55.76, 287.92) mm, rotated rx -18.18 ry -0.39 rz 0.13 deg; joints [20.747, -106.003, -119.144, -33.336, 87.264, 15.093]
  MoveL 519 to (-135.07, 65.31, 284.92) mm, rotated rx -17.77 ry -0.33 rz 0.1 deg; joints [21.163, -105.046, -121.167, -31.911, 87.007, 15.479]
  MoveL 520 to (-135.08, 74.92, 281.94) mm, rotated rx -17.34 ry -0.29 rz 0.09 deg; joints [21.596, -104.102, -123.197, -30.443, 86.762, 15.879]
  MoveL 521 to (-135.04, 81.73, 280) mm, rotated rx -17.18 ry -0.26 rz 0.08 deg; joints [21.882, -103.496, -124.494, -29.62, 86.629, 16.149]
  MoveL 522 to (-135.03, 86.92, 278.05) mm, rotated rx -17.18 ry -0.15 rz 0.04 deg; joints [22.16, -102.981, -125.383, -29.292, 86.451, 16.423]
  MoveL 523 to (-135.03, 94.88, 275.6) mm, rotated rx -16.99 ry -0.14 rz 0.04 deg; joints [22.508, -102.253, -126.885, -28.368, 86.316, 16.752]
  MoveL 524 to (-135.05, 104.86, 273.09) mm, rotated rx -16.64 ry -0.22 rz 0.07 deg; joints [22.915, -101.425, -128.852, -26.892, 86.209, 17.125]
  MoveL 525 to (-137.85, 110.55, 271) mm, rotated rx -16.34 ry -0.13 rz 0.04 deg; joints [23.659, -100.831, -130.045, -26.083, 85.857, 17.833]
  MoveL 526 to (-125.01, -254.46, 398.5) mm, rotated rx -16.58 ry -0.88 rz 0.26 deg; joints [13.827, -141.096, -50.982, -64.497, 88.939, 8.257]
  MoveL 527 to (-124.95, -245.96, 396.76) mm, rotated rx -18.91 ry -1.12 rz 0.38 deg; joints [13.685, -141.5, -49.71, -67.634, 89.562, 8.192]
  MoveL 528 to (-125.11, -236.29, 394.25) mm, rotated rx -20.94 ry -1.23 rz 0.47 deg; joints [13.637, -141.482, -49.389, -69.956, 89.992, 8.196]
  MoveL 529 to (-125.03, -228.27, 391.19) mm, rotated rx -21.78 ry -1.02 rz 0.41 deg; joints [13.753, -140.719, -50.696, -70.283, 89.881, 8.33]
  MoveL 530 to (-125.21, -222.32, 387.85) mm, rotated rx -22.72 ry -0.7 rz 0.29 deg; joints [13.916, -140.286, -51.168, -71.226, 89.653, 8.51]
  MoveL 531 to (-124.82, -214.75, 384.39) mm, rotated rx -23.12 ry -0.14 rz 0.06 deg; joints [14.181, -139.224, -53.085, -70.859, 89.085, 8.782]
  MoveL 532 to (-125.38, -207.05, 381.37) mm, rotated rx -22.33 ry -0.02 rz 0.01 deg; joints [14.409, -137.375, -56.919, -68.121, 88.806, 8.992]
  MoveL 533 to (-124.76, -201.34, 379) mm, rotated rx -21.69 ry 0.09 rz -0.04 deg; joints [14.521, -136.025, -59.712, -66.07, 88.57, 9.09]
  MoveL 534 to (-125.18, -194.45, 377.05) mm, rotated rx -20.87 ry 0.03 rz -0.01 deg; joints [14.659, -134.547, -62.947, -63.494, 88.487, 9.207]
  MoveL 535 to (-124.88, -184.37, 372.52) mm, rotated rx -20.4 ry -0.23 rz 0.09 deg; joints [14.693, -132.75, -66.52, -61.21, 88.678, 9.227]
  MoveL 536 to (-126.22, -178.24, 370) mm, rotated rx -20.39 ry -0.66 rz 0.24 deg; joints [14.695, -131.878, -68.232, -60.281, 89.126, 9.226]
  MoveL 537 to (-124.69, -174.11, 368.4) mm, rotated rx -20.52 ry -0.92 rz 0.34 deg; joints [14.511, -131.384, -69.176, -59.912, 89.452, 9.048]
  MoveL 538 to (-125.08, -164.71, 365.8) mm, rotated rx -20.71 ry -1.21 rz 0.46 deg; joints [14.517, -130.347, -71.329, -58.936, 89.794, 9.059]
  MoveL 539 to (-124.69, -154.85, 362.07) mm, rotated rx -20.18 ry -0.82 rz 0.3 deg; joints [14.829, -128.785, -74.507, -56.87, 89.242, 9.353]
  MoveL 540 to (-128.1, -150.42, 359) mm, rotated rx -19.55 ry -0.55 rz 0.19 deg; joints [15.339, -127.759, -76.448, -55.392, 88.758, 9.837]
  MoveL 541 to (-125.28, -144.88, 357.52) mm, rotated rx -19.42 ry -0.33 rz 0.12 deg; joints [15.3, -127.069, -77.919, -54.524, 88.513, 9.796]
  MoveL 542 to (-124.81, -135.39, 354.72) mm, rotated rx -19.95 ry 0.09 rz -0.03 deg; joints [15.553, -126.237, -79.484, -54.391, 88.116, 10.063]
  MoveL 543 to (-124.97, -125.37, 351.77) mm, rotated rx -20.47 ry 0.61 rz -0.23 deg; joints [15.912, -125.362, -81.139, -54.233, 87.609, 10.437]
  MoveL 544 to (-127.23, -118.8, 350) mm, rotated rx -20.89 ry 0.95 rz -0.36 deg; joints [16.323, -124.86, -82.092, -54.279, 87.265, 10.859]
  MoveL 545 to (-124.83, -113.95, 347.05) mm, rotated rx -20.78 ry 0.66 rz -0.25 deg; joints [16.089, -124.099, -83.415, -53.541, 87.585, 10.621]
  MoveL 546 to (-124.85, -104.42, 342.64) mm, rotated rx -20.36 ry 0.16 rz -0.06 deg; joints [16.057, -122.712, -86.089, -51.745, 88.034, 10.573]
  MoveL 547 to (-124.74, -97.23, 340) mm, rotated rx -19.85 ry -0.12 rz 0.04 deg; joints [16.078, -121.689, -88.234, -50.075, 88.228, 10.577]
  MoveL 548 to (-125.13, -92.57, 338.61) mm, rotated rx -19.69 ry -0.12 rz 0.04 deg; joints [16.204, -121.138, -89.408, -49.29, 88.176, 10.695]
  MoveL 549 to (-125.08, -84.98, 337.44) mm, rotated rx -19.64 ry -0.06 rz 0.02 deg; joints [16.353, -120.472, -90.994, -48.338, 88.081, 10.84]
  MoveL 550 to (-124.93, -75.06, 332.82) mm, rotated rx -19.69 ry -0.07 rz 0.02 deg; joints [16.519, -119.293, -93.063, -47.503, 88.07, 11.005]
  MoveL 551 to (-124.26, -68.72, 330.11) mm, rotated rx -19.53 ry 0.02 rz -0.01 deg; joints [16.641, -118.497, -94.563, -46.661, 87.924, 11.121]
  MoveL 552 to (-124.99, -63.68, 328.04) mm, rotated rx -19.73 ry 0.07 rz -0.03 deg; joints [16.811, -118.009, -95.382, -46.547, 87.882, 11.296]
  MoveL 553 to (-125.23, -55.25, 324.94) mm, rotated rx -19.94 ry 0.07 rz -0.03 deg; joints [16.979, -117.189, -96.872, -46.087, 87.892, 11.469]
  MoveL 554 to (-124.98, -44.83, 322.12) mm, rotated rx -19.76 ry -0.04 rz 0.01 deg; joints [17.114, -116.153, -99.095, -44.711, 87.952, 11.594]
  MoveL 555 to (-125.99, -38.05, 320) mm, rotated rx -19.6 ry -0.18 rz 0.06 deg; joints [17.29, -115.441, -100.579, -43.759, 88.031, 11.761]
  MoveL 556 to (-125.07, -33.48, 318.04) mm, rotated rx -19.38 ry -0.25 rz 0.09 deg; joints [17.286, -114.853, -101.719, -42.967, 88.063, 11.748]
  MoveL 557 to (-124.8, -25.36, 314.48) mm, rotated rx -19.23 ry -0.4 rz 0.14 deg; joints [17.376, -113.898, -103.465, -42.004, 88.17, 11.83]
  MoveL 558 to (-124.94, -15.73, 311.22) mm, rotated rx -18.92 ry -0.46 rz 0.16 deg; joints [17.601, -112.851, -105.605, -40.597, 88.129, 12.038]
  MoveL 559 to (-125.13, -5, 307.66) mm, rotated rx -18.06 ry -0.39 rz 0.13 deg; joints [18.008, -111.554, -108.431, -38.262, 87.788, 12.401]
  MoveL 560 to (-125.13, 5.22, 304.3) mm, rotated rx -16.92 ry -0.36 rz 0.11 deg; joints [18.413, -110.27, -111.382, -35.506, 87.424, 12.744]
  MoveL 561 to (-125.11, 14.72, 301.49) mm, rotated rx -16.83 ry -0.64 rz 0.19 deg; joints [18.497, -109.418, -113.188, -34.396, 87.669, 12.818]
  MoveL 562 to (-124.58, 21.3, 300) mm, rotated rx -17.11 ry -0.68 rz 0.21 deg; joints [18.539, -108.98, -114.086, -34.203, 87.766, 12.873]
  MoveL 563 to (-125.22, 26.48, 298.07) mm, rotated rx -17.86 ry -0.57 rz 0.18 deg; joints [18.718, -108.662, -114.32, -35.051, 87.777, 13.086]
  MoveL 564 to (-125.11, 35.38, 295.67) mm, rotated rx -18.81 ry -0.3 rz 0.1 deg; joints [18.972, -108.166, -114.994, -35.881, 87.672, 13.382]
  MoveL 565 to (-125.01, 45.47, 292) mm, rotated rx -19.01 ry -0.37 rz 0.13 deg; joints [19.174, -107.24, -116.617, -35.367, 87.752, 13.589]
  MoveL 566 to (-127.35, 51.3, 290) mm, rotated rx -18.68 ry -0.4 rz 0.14 deg; joints [19.632, -106.609, -117.937, -34.369, 87.623, 14.023]
  MoveL 567 to (-124.78, 55.85, 288.05) mm, rotated rx -18.3 ry -0.36 rz 0.12 deg; joints [19.569, -106.012, -119.115, -33.42, 87.494, 13.943]
  MoveL 568 to (-125.12, 65.43, 285.14) mm, rotated rx -17.78 ry -0.27 rz 0.09 deg; joints [20.035, -105.043, -121.233, -31.814, 87.184, 14.375]
  MoveL 569 to (-125.01, 74.95, 281.77) mm, rotated rx -17.37 ry -0.33 rz 0.1 deg; joints [20.363, -104.048, -123.253, -30.389, 87.071, 14.673]
  MoveL 570 to (-124.9, 81.48, 280.24) mm, rotated rx -17.25 ry -0.3 rz 0.09 deg; joints [20.596, -103.53, -124.452, -29.615, 86.967, 14.895]
  MoveL 571 to (-125.11, 86.63, 278.04) mm, rotated rx -17.13 ry -0.45 rz 0.14 deg; joints [20.731, -102.966, -125.459, -29.021, 87.054, 15.018]
  MoveL 572 to (-124.92, 94.7, 275.56) mm, rotated rx -16.85 ry -0.63 rz 0.19 deg; joints [20.919, -102.222, -127.077, -27.832, 87.118, 15.182]
  MoveL 573 to (-125.06, 104.02, 272.9) mm, rotated rx -16.2 ry -0.75 rz 0.22 deg; joints [21.317, -101.344, -129.204, -25.945, 86.972, 15.528]
  MoveL 574 to (-112.18, -256.58, 400) mm, rotated rx -14.52 ry -0.79 rz 0.21 deg; joints [13.038, -140.122, -53.719, -60.694, 88.751, 7.421]
  MoveL 575 to (-115.43, -253.18, 399) mm, rotated rx -15.63 ry -0.83 rz 0.23 deg; joints [13.23, -140.32, -52.991, -62.321, 88.895, 7.645]
  MoveL 576 to (-114.97, -244.48, 397.18) mm, rotated rx -18.69 ry -0.54 rz 0.18 deg; joints [13.236, -141.168, -50.549, -66.993, 89.008, 7.746]
  MoveL 577 to (-115.27, -235.13, 394.03) mm, rotated rx -20.97 ry -0.49 rz 0.19 deg; joints [13.252, -141.311, -49.712, -69.954, 89.272, 7.817]
  MoveL 578 to (-114.64, -228.4, 391.33) mm, rotated rx -22.26 ry -0.32 rz 0.13 deg; joints [13.279, -141.116, -49.766, -71.4, 89.265, 7.87]
  MoveL 579 to (-115.54, -222.77, 388.44) mm, rotated rx -23.28 ry -0.1 rz 0.05 deg; joints [13.437, -140.84, -49.973, -72.508, 89.158, 8.046]
  MoveL 580 to (-115.22, -214.61, 384.92) mm, rotated rx -23.35 ry 0.12 rz -0.05 deg; joints [13.591, -139.423, -52.714, -71.291, 88.908, 8.201]
  MoveL 581 to (-115.03, -205.74, 381.53) mm, rotated rx -22.43 ry 0.07 rz -0.03 deg; joints [13.707, -137.286, -57.166, -68.059, 88.813, 8.299]
  MoveL 582 to (-114.29, -200.4, 379) mm, rotated rx -21.74 ry 0.15 rz -0.06 deg; joints [13.789, -135.932, -59.934, -65.98, 88.616, 8.367]
  MoveL 583 to (-115.06, -194.4, 376.41) mm, rotated rx -20.83 ry 0.25 rz -0.09 deg; joints [14.009, -134.418, -63.11, -63.43, 88.352, 8.564]
  MoveL 584 to (-115.11, -184.47, 373.1) mm, rotated rx -19.99 ry 0.17 rz -0.06 deg; joints [14.15, -132.568, -67.06, -60.499, 88.28, 8.682]
  MoveL 585 to (-113.68, -176.97, 370.24) mm, rotated rx -19.62 ry 0.08 rz -0.03 deg; joints [14.117, -131.338, -69.586, -58.822, 88.328, 8.639]
  MoveL 586 to (-116.41, -173.31, 368.86) mm, rotated rx -19.99 ry -0.39 rz 0.14 deg; joints [14.145, -131.055, -70.061, -58.916, 88.878, 8.674]
  MoveL 587 to (-114.97, -165.01, 366.22) mm, rotated rx -20.71 ry -0.55 rz 0.21 deg; joints [14.021, -130.399, -71.231, -59.092, 89.172, 8.571]
  MoveL 588 to (-115.12, -154.84, 362.46) mm, rotated rx -20.43 ry -0.59 rz 0.22 deg; joints [14.16, -128.939, -74.185, -57.313, 89.154, 8.7]
  MoveL 589 to (-112.93, -148.96, 360) mm, rotated rx -20.06 ry -0.55 rz 0.2 deg; joints [14.106, -127.981, -76.121, -55.977, 89.063, 8.638]
  MoveL 590 to (-115.5, -144.7, 357.46) mm, rotated rx -19.71 ry -0.47 rz 0.17 deg; joints [14.434, -127.172, -77.643, -54.933, 88.864, 8.951]
  MoveL 591 to (-114.95, -135.27, 354) mm, rotated rx -20.14 ry -0.54 rz 0.2 deg; joints [14.458, -126.234, -79.356, -54.578, 88.999, 8.987]
  MoveL 592 to (-114.97, -126.13, 351.49) mm, rotated rx -20.98 ry -0.49 rz 0.19 deg; joints [14.545, -125.626, -80.446, -54.931, 89.066, 9.094]
  MoveL 593 to (-114.96, -120.69, 349) mm, rotated rx -21.1 ry -0.43 rz 0.17 deg; joints [14.64, -124.978, -81.587, -54.567, 89.011, 9.192]
  MoveL 594 to (-115.03, -115.3, 346.48) mm, rotated rx -20.81 ry -0.41 rz 0.15 deg; joints [14.759, -124.145, -83.193, -53.512, 88.92, 9.302]
  MoveL 595 to (-114.98, -104.97, 342.68) mm, rotated rx -19.99 ry -0.29 rz 0.11 deg; joints [15.023, -122.591, -86.435, -51.044, 88.622, 9.54]
  MoveL 596 to (-115.1, -98.03, 340) mm, rotated rx -19.55 ry -0.36 rz 0.13 deg; joints [15.143, -121.608, -88.452, -49.562, 88.6, 9.644]
  MoveL 597 to (-114.81, -93.09, 338.46) mm, rotated rx -19.4 ry -0.6 rz 0.21 deg; joints [15.088, -121.038, -89.662, -48.738, 88.834, 9.585]
  MoveL 598 to (-115.04, -84.57, 335.93) mm, rotated rx -19.5 ry -1 rz 0.35 deg; joints [15.034, -120.221, -91.342, -47.896, 89.277, 9.534]
  MoveL 599 to (-114.96, -74.96, 332.39) mm, rotated rx -20.08 ry -0.81 rz 0.3 deg; joints [15.227, -119.395, -92.724, -47.953, 89.147, 9.742]
  MoveL 600 to (-115.18, -67.69, 330.47) mm, rotated rx -19.94 ry -0.44 rz 0.16 deg; joints [15.561, -118.634, -94.338, -47.036, 88.676, 10.068]
  MoveL 601 to (-115.18, -62.15, 328.06) mm, rotated rx -19.92 ry -0.22 rz 0.08 deg; joints [15.774, -117.978, -95.513, -46.538, 88.406, 10.279]
  MoveL 602 to (-114.91, -54.58, 324.65) mm, rotated rx -19.79 ry -0.23 rz 0.08 deg; joints [15.898, -117.048, -97.207, -45.649, 88.368, 10.396]
  MoveL 603 to (-114.93, -44.84, 321.71) mm, rotated rx -19.56 ry -0.23 rz 0.08 deg; joints [16.096, -116.019, -99.356, -44.312, 88.29, 10.583]
  MoveL 604 to (-114.98, -35.16, 317.82) mm, rotated rx -19.28 ry -0.43 rz 0.15 deg; joints [16.209, -114.878, -101.56, -42.936, 88.424, 10.684]
  MoveL 605 to (-115, -25.7, 314.97) mm, rotated rx -19.11 ry -0.6 rz 0.21 deg; joints [16.312, -113.936, -103.533, -41.708, 88.555, 10.778]
  MoveL 606 to (-114.91, -15.77, 311.43) mm, rotated rx -18.89 ry -0.55 rz 0.19 deg; joints [16.558, -112.866, -105.638, -40.477, 88.407, 11.012]
  MoveL 607 to (-115.15, -5.03, 307.73) mm, rotated rx -18.15 ry -0.77 rz 0.25 deg; joints [16.762, -111.596, -108.371, -38.245, 88.45, 11.182]
  MoveL 608 to (-115.05, 5.39, 304.2) mm, rotated rx -16.87 ry -0.75 rz 0.23 deg; joints [17.134, -110.242, -111.497, -35.233, 88.099, 11.49]
  MoveL 609 to (-115.03, 14.73, 301.57) mm, rotated rx -16.71 ry -0.62 rz 0.19 deg; joints [17.444, -109.39, -113.317, -34.147, 87.856, 11.785]
  MoveL 610 to (-115.29, 22.61, 300) mm, rotated rx -17.45 ry -0.49 rz 0.16 deg; joints [17.633, -108.992, -114.008, -34.61, 87.843, 12.006]
  MoveL 611 to (-115.03, 27.74, 298.7) mm, rotated rx -18.16 ry -0.43 rz 0.14 deg; joints [17.675, -108.76, -114.254, -35.306, 87.92, 12.079]
  MoveL 612 to (-115.09, 35.27, 295.49) mm, rotated rx -18.95 ry -0.45 rz 0.15 deg; joints [17.765, -108.18, -114.885, -36.033, 88.089, 12.201]
  MoveL 613 to (-114.98, 45.47, 291.57) mm, rotated rx -19.02 ry -0.17 rz 0.06 deg; joints [18.184, -107.159, -116.649, -35.435, 87.737, 12.618]
  MoveL 614 to (-115.1, 55.49, 288.19) mm, rotated rx -18.37 ry -0.07 rz 0.02 deg; joints [18.621, -106.044, -119.006, -33.601, 87.407, 13.02]
  MoveL 615 to (-115.14, 65.32, 285.22) mm, rotated rx -17.7 ry -0.23 rz 0.07 deg; joints [18.899, -105.029, -121.313, -31.633, 87.357, 13.259]
  MoveL 616 to (-115.14, 75.14, 282.9) mm, rotated rx -17.35 ry -0.34 rz 0.11 deg; joints [19.16, -104.208, -123.294, -30.112, 87.333, 13.496]
  MoveL 617 to (-115, 83.01, 280.58) mm, rotated rx -16.98 ry -0.54 rz 0.16 deg; joints [19.306, -103.479, -124.958, -28.779, 87.417, 13.617]
  MoveL 618 to (-115.28, 87.98, 278.23) mm, rotated rx -16.93 ry -0.5 rz 0.15 deg; joints [19.547, -102.905, -125.869, -28.415, 87.31, 13.85]
  MoveL 619 to (-115.12, 94.91, 276.01) mm, rotated rx -16.87 ry -0.53 rz 0.16 deg; joints [19.741, -102.282, -127.102, -27.738, 87.288, 14.035]
  MoveL 620 to (-115.11, 102.86, 273.37) mm, rotated rx -16.63 ry -0.67 rz 0.2 deg; joints [19.958, -101.533, -128.651, -26.687, 87.317, 14.232]
  MoveL 621 to (-103.58, -255.61, 399) mm, rotated rx -15.18 ry 0.1 rz -0.03 deg; joints [12.755, -140.308, -52.991, -62.004, 87.993, 7.174]
  MoveL 622 to (-105.86, -254.01, 400.11) mm, rotated rx -15.7 ry -0.06 rz 0.02 deg; joints [12.838, -140.591, -52.506, -62.705, 88.2, 7.271]
  MoveL 623 to (-98.47, -251.93, 400) mm, rotated rx -16.86 ry 0.45 rz -0.14 deg; joints [12.477, -141.122, -51.157, -64.728, 87.904, 6.956]
  MoveL 624 to (-99.34, -249.14, 400) mm, rotated rx -17.71 ry 0.45 rz -0.14 deg; joints [12.522, -141.375, -50.544, -65.934, 87.995, 7.023]
  MoveL 625 to (-103, -249.14, 400) mm, rotated rx -17.36 ry 0.35 rz -0.11 deg; joints [12.755, -141.117, -51.167, -65.217, 88.011, 7.241]
  MoveL 626 to (-105.47, -244.29, 397.97) mm, rotated rx -18.83 ry 0.32 rz -0.11 deg; joints [12.899, -141.324, -50.296, -67.337, 88.188, 7.422]
  MoveL 627 to (-104.93, -235.1, 394.1) mm, rotated rx -20.91 ry 0.36 rz -0.14 deg; joints [12.868, -141.252, -49.83, -69.945, 88.422, 7.439]
  MoveL 628 to (-105.03, -228.13, 390.95) mm, rotated rx -22.39 ry 0.15 rz -0.06 deg; joints [12.789, -141.129, -49.655, -71.682, 88.849, 7.388]
  MoveL 629 to (-105.1, -222.02, 387.42) mm, rotated rx -23.48 ry -0.11 rz 0.05 deg; joints [12.7, -140.785, -49.935, -72.791, 89.28, 7.317]
  MoveL 630 to (-105.37, -214.69, 384.15) mm, rotated rx -23.36 ry -0.09 rz 0.04 deg; joints [12.808, -139.352, -52.746, -71.295, 89.229, 7.422]
  MoveL 631 to (-104.87, -206.93, 381.25) mm, rotated rx -22.63 ry -0.06 rz 0.02 deg; joints [12.9, -137.536, -56.523, -68.616, 89.085, 7.502]
  MoveL 632 to (-103.54, -202.38, 379) mm, rotated rx -21.96 ry -0.22 rz 0.09 deg; joints [12.817, -136.305, -59.051, -66.632, 89.187, 7.407]
  MoveL 633 to (-105.19, -195.45, 376.05) mm, rotated rx -21.04 ry -0.01 rz 0.01 deg; joints [13.148, -134.624, -62.545, -63.944, 88.791, 7.718]
  MoveL 634 to (-104.94, -185.13, 372.87) mm, rotated rx -20.13 ry 0.26 rz -0.09 deg; joints [13.403, -132.682, -66.722, -60.851, 88.341, 7.95]
  MoveL 635 to (-105.39, -176.73, 370.3) mm, rotated rx -19.53 ry 0.53 rz -0.19 deg; joints [13.683, -131.267, -69.761, -58.686, 87.921, 8.211]
  MoveL 636 to (-104.3, -172.49, 368.93) mm, rotated rx -19.47 ry 0.55 rz -0.2 deg; joints [13.661, -130.694, -70.942, -58.017, 87.894, 8.188]
  MoveL 637 to (-105.07, -164.63, 365.69) mm, rotated rx -20.43 ry 0.32 rz -0.12 deg; joints [13.659, -130.137, -71.725, -58.707, 88.273, 8.21]
  MoveL 638 to (-105.18, -154.72, 362.48) mm, rotated rx -20.24 ry -0.05 rz 0.02 deg; joints [13.632, -128.823, -74.451, -57.047, 88.642, 8.176]
  MoveL 639 to (-105.79, -148.95, 360.69) mm, rotated rx -19.91 ry -0.18 rz 0.06 deg; joints [13.711, -127.977, -76.269, -55.731, 88.716, 8.246]
  MoveL 640 to (-104.69, -143.84, 357.46) mm, rotated rx -19.56 ry -0.3 rz 0.11 deg; joints [13.659, -127.031, -78.013, -54.565, 88.806, 8.186]
  MoveL 641 to (-104.87, -135.51, 354.09) mm, rotated rx -19.95 ry -0.46 rz 0.17 deg; joints [13.682, -126.173, -79.533, -54.266, 89.024, 8.218]
  MoveL 642 to (-104.92, -126.08, 351.3) mm, rotated rx -20.75 ry -0.63 rz 0.24 deg; joints [13.675, -125.501, -80.736, -54.504, 89.316, 8.229]
  MoveL 643 to (-105.38, -120.69, 349) mm, rotated rx -20.79 ry -0.85 rz 0.32 deg; joints [13.674, -124.852, -81.949, -53.946, 89.561, 8.229]
  MoveL 644 to (-99.9, -120.69, 349) mm, rotated rx -20.48 ry -0.94 rz 0.35 deg; joints [13.2, -124.725, -82.293, -53.407, 89.685, 7.755]
  MoveL 645 to (-105.08, -115.41, 346.89) mm, rotated rx -20.72 ry -1.13 rz 0.43 deg; joints [13.59, -124.191, -83.243, -53.198, 89.86, 8.145]
  MoveL 646 to (-105.11, -105, 342.78) mm, rotated rx -20.23 ry -1.12 rz 0.41 deg; joints [13.766, -122.74, -86.151, -51.258, 89.749, 8.307]
  MoveL 647 to (-104.6, -96.04, 340.31) mm, rotated rx -19.36 ry -1.08 rz 0.38 deg; joints [13.922, -121.463, -89.034, -48.796, 89.54, 8.437]
  MoveL 648 to (-106.16, -91.67, 338.85) mm, rotated rx -19.1 ry -0.88 rz 0.31 deg; joints [14.234, -120.885, -90.245, -47.947, 89.237, 8.736]
  MoveL 649 to (-98.37, -90.65, 339) mm, rotated rx -19.15 ry -1.2 rz 0.42 deg; joints [13.4, -120.888, -90.349, -47.833, 89.736, 7.918]
  MoveL 650 to (-105.11, -84.5, 335.39) mm, rotated rx -19.32 ry -0.95 rz 0.33 deg; joints [14.201, -120.087, -91.567, -47.623, 89.346, 8.71]
  MoveL 651 to (-104.91, -74.85, 332.17) mm, rotated rx -20.25 ry -1.2 rz 0.44 deg; joints [14.123, -119.451, -92.571, -48.129, 89.774, 8.659]
  MoveL 652 to (-104.77, -68.21, 330.2) mm, rotated rx -20.35 ry -1.14 rz 0.42 deg; joints [14.232, -118.825, -93.818, -47.622, 89.7, 8.769]
  MoveL 653 to (-105.09, -62.79, 328.24) mm, rotated rx -20.13 ry -1.02 rz 0.37 deg; joints [14.419, -118.156, -95.162, -46.752, 89.512, 8.946]
  MoveL 654 to (-104.8, -54.62, 324.9) mm, rotated rx -19.8 ry -0.97 rz 0.35 deg; joints [14.575, -117.12, -97.174, -45.462, 89.377, 9.091]
  MoveL 655 to (-104.96, -44.92, 321.87) mm, rotated rx -19.63 ry -0.92 rz 0.33 deg; joints [14.781, -116.102, -99.265, -44.228, 89.262, 9.289]
  MoveL 656 to (-104.97, -35.14, 317.68) mm, rotated rx -19.11 ry -0.91 rz 0.31 deg; joints [15.004, -114.83, -101.733, -42.528, 89.117, 9.493]
  MoveL 657 to (-104.98, -25.85, 315.78) mm, rotated rx -19.13 ry -0.91 rz 0.31 deg; joints [15.154, -114.077, -103.448, -41.59, 89.092, 9.64]
  MoveL 658 to (-104.95, -15.58, 311.77) mm, rotated rx -18.77 ry -0.94 rz 0.32 deg; joints [15.354, -112.888, -105.774, -40.093, 89.028, 9.824]
  MoveL 659 to (-103.32, -9.33, 310) mm, rotated rx -18.05 ry -1.22 rz 0.4 deg; joints [15.211, -112.129, -107.619, -38.246, 89.222, 9.659]
  MoveL 660 to (-105.42, -4.33, 307.62) mm, rotated rx -17.81 ry -1.21 rz 0.39 deg; joints [15.56, -111.48, -108.815, -37.468, 89.087, 9.991]
  MoveL 661 to (-105.05, 5.3, 304.64) mm, rotated rx -17.05 ry -1.08 rz 0.33 deg; joints [15.858, -110.385, -111.291, -35.367, 88.758, 10.253]
  MoveL 662 to (-104.94, 14.75, 302.21) mm, rotated rx -17.16 ry -0.85 rz 0.26 deg; joints [16.16, -109.619, -112.874, -34.71, 88.474, 10.552]
  MoveL 663 to (-104.59, 22.05, 300.19) mm, rotated rx -17.56 ry -0.61 rz 0.19 deg; joints [16.379, -109.091, -113.799, -34.763, 88.25, 10.784]
  MoveL 664 to (-105.29, 27.23, 298.2) mm, rotated rx -17.99 ry -0.62 rz 0.2 deg; joints [16.514, -108.686, -114.341, -35.049, 88.319, 10.934]
  MoveL 665 to (-105.11, 35.31, 295.33) mm, rotated rx -18.98 ry -0.59 rz 0.2 deg; joints [16.585, -108.181, -114.866, -36.016, 88.461, 11.042]
  MoveL 666 to (-105.46, 44.81, 291.92) mm, rotated rx -19.45 ry -0.42 rz 0.15 deg; joints [16.895, -107.381, -116.136, -36.043, 88.321, 11.365]
  MoveL 667 to (-102.87, 49.11, 289) mm, rotated rx -19.02 ry -0.49 rz 0.17 deg; joints [16.727, -106.652, -117.338, -35.13, 88.344, 11.183]
  MoveL 668 to (-99.35, 49.61, 289) mm, rotated rx -18.97 ry -0.74 rz 0.25 deg; joints [16.189, -106.642, -117.453, -34.912, 88.688, 10.652]
  MoveL 669 to (-105, 55.38, 287.96) mm, rotated rx -18.15 ry -0.44 rz 0.15 deg; joints [17.251, -105.987, -119.204, -33.101, 88.016, 11.663]
  MoveL 670 to (-105.07, 65.32, 285.06) mm, rotated rx -17.69 ry -0.44 rz 0.14 deg; joints [17.573, -105.027, -121.332, -31.499, 87.849, 11.959]
  MoveL 671 to (-104.94, 74.93, 282) mm, rotated rx -17.13 ry -0.47 rz 0.14 deg; joints [17.876, -104.047, -123.488, -29.775, 87.696, 12.228]
  MoveL 672 to (-105.03, 81, 280) mm, rotated rx -16.9 ry -0.61 rz 0.19 deg; joints [17.993, -103.464, -124.726, -28.872, 87.768, 12.33]
  MoveL 673 to (-104.97, 86.36, 278.54) mm, rotated rx -16.93 ry -0.63 rz 0.19 deg; joints [18.122, -103.04, -125.597, -28.461, 87.76, 12.457]
  MoveL 674 to (-105.13, 95.31, 275.93) mm, rotated rx -16.77 ry -0.6 rz 0.18 deg; joints [18.447, -102.26, -127.253, -27.438, 87.628, 12.766]
  MoveL 675 to (-104.94, 103.18, 274.19) mm, rotated rx -16.1 ry -0.66 rz 0.19 deg; joints [18.72, -101.593, -129.13, -25.578, 87.473, 12.996]
  MoveL 676 to (-94.29, -254.03, 398.79) mm, rotated rx -17.02 ry 0.4 rz -0.12 deg; joints [12.145, -141.384, -50.293, -65.473, 88.049, 6.637]
  MoveL 677 to (-95.02, -244.65, 397.59) mm, rotated rx -19.41 ry 0.37 rz -0.13 deg; joints [12.154, -141.789, -49.132, -68.594, 88.354, 6.703]
  MoveL 678 to (-94.68, -235.48, 393.84) mm, rotated rx -20.94 ry 0.35 rz -0.13 deg; joints [12.139, -141.312, -49.65, -70.072, 88.554, 6.719]
  MoveL 679 to (-95.64, -228.25, 390.76) mm, rotated rx -21.64 ry 0.04 rz -0.02 deg; joints [12.118, -140.552, -50.958, -70.187, 88.966, 6.711]
  MoveL 680 to (-94.68, -222.63, 387.7) mm, rotated rx -22.79 ry -0.54 rz 0.23 deg; joints [11.818, -140.379, -50.925, -71.458, 89.762, 6.43]
  MoveL 681 to (-94.68, -214.92, 384.12) mm, rotated rx -23.17 ry -1.12 rz 0.48 deg; joints [11.631, -139.29, -52.946, -70.831, 90.458, 6.25]
  MoveL 682 to (-94.97, -207.14, 381.07) mm, rotated rx -22.53 ry -1.21 rz 0.5 deg; joints [11.711, -137.524, -56.593, -68.296, 90.465, 6.321]
  MoveL 683 to (-95.62, -202.38, 379) mm, rotated rx -21.98 ry -1.13 rz 0.45 deg; joints [11.861, -136.365, -58.976, -66.539, 90.289, 6.46]
  MoveL 684 to (-95, -195.95, 376.1) mm, rotated rx -21.54 ry -1.06 rz 0.42 deg; joints [11.925, -135.051, -61.61, -64.795, 90.152, 6.516]
  MoveL 685 to (-95.09, -185.24, 372.31) mm, rotated rx -20.62 ry -0.5 rz 0.19 deg; joints [12.312, -132.952, -66.004, -61.659, 89.386, 6.882]
